REGION Network 7: Отключение
   RUNG wire#powerrail
      I_Contact( #Use.QF )
      wire#w1
      Coil( #xQF )
   END_RUNG
   RUNG wire#powerrail
      Contact( #CMD.Sim )
   END_RUNG wire#w1
   RUNG wire#powerrail
      Contact( #Use.QF )
      Contact( #FB.QF )
      I_Contact( #CMD.Sim )
   END_RUNG wire#w1
   RUNG wire#powerrail
      I_Contact( #Use.KM )
      Contact( #CMD.Start_M )
      I_Contact( #CMD.Sim )
      wire#w2
      Coil( #xKM )
   END_RUNG
   RUNG wire#powerrail
      Contact( #Use.KM )
      wire#w3
      Contact( #FB.KM )
   END_RUNG wire#w2
   RUNG wire#powerrail
      Contact( #CMD.Sim )
   END_RUNG wire#w3
   // the same network as SCL:
   #xQF := NOT #Use.QF OR #CMD.Sim OR (#Use.QF AND #FB.QF AND NOT #CMD.Sim);
   #xKM := (NOT #Use.KM AND #CMD.Start_M AND NOT #CMD.Sim) OR ((#Use.KM OR #CMD.Sim) AND #FB.KM);
END_REGION

REGION Network 8: Режим работы устройства / определение режима работы
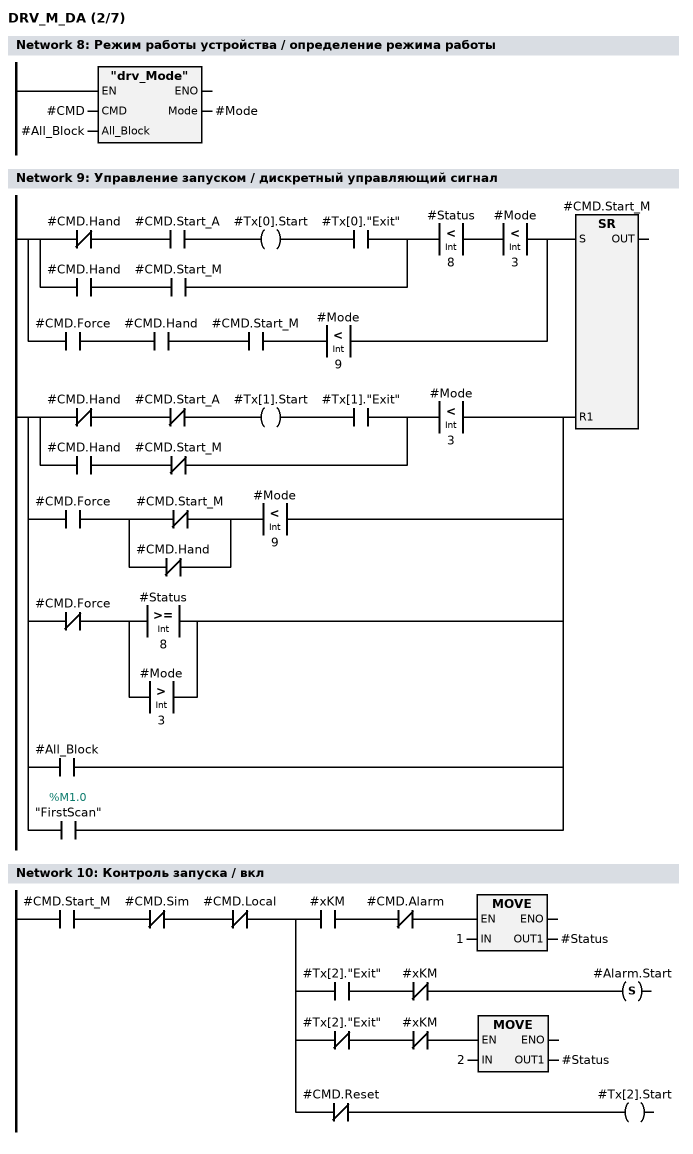
   RUNG wire#powerrail
      "drv_Mode"(CMD := #CMD, All_Block := #All_Block, Mode => #Mode)
   END_RUNG
   // the same network as SCL:
   "drv_Mode"(CMD := #CMD, All_Block := #All_Block, Mode => #Mode);
END_REGION

REGION Network 9: Управление запуском / дискретный управляющий сигнал
   RUNG wire#powerrail
      I_Contact( #CMD.Hand )
      Contact( #CMD.Start_A )
      Coil( #Tx[0].Start )
      Contact( #Tx[0]."Exit" )
      wire#w1
      { S7_Templates := "SrcType := Int" } LT_Contact(in1 := #Status, in2 := 8)
      { S7_Templates := "SrcType := Int" } LT_Contact(in1 := #Mode, in2 := 3)
      wire#w2
      S_SR(operand := #CMD.Start_M, r1 := wire#w7)
   END_RUNG
   RUNG wire#powerrail
      Contact( #CMD.Hand )
      Contact( #CMD.Start_M )
   END_RUNG wire#w1
   RUNG wire#powerrail
      Contact( #CMD.Force )
      Contact( #CMD.Hand )
      Contact( #CMD.Start_M )
      { S7_Templates := "SrcType := Int" } LT_Contact(in1 := #Mode, in2 := 9)
   END_RUNG wire#w2
   RUNG wire#powerrail
      I_Contact( #CMD.Hand )
      I_Contact( #CMD.Start_A )
      Coil( #Tx[1].Start )
      Contact( #Tx[1]."Exit" )
      wire#w3
      { S7_Templates := "SrcType := Int" } LT_Contact(in1 := #Mode, in2 := 3)
   END_RUNG wire#w7
   RUNG wire#powerrail
      Contact( #CMD.Hand )
      I_Contact( #CMD.Start_M )
   END_RUNG wire#w3
   RUNG wire#powerrail
      Contact( #CMD.Force )
      wire#w4
      I_Contact( #CMD.Start_M )
      wire#w5
      { S7_Templates := "SrcType := Int" } LT_Contact(in1 := #Mode, in2 := 9)
   END_RUNG wire#w7
   RUNG wire#w4
      I_Contact( #CMD.Hand )
   END_RUNG wire#w5
   RUNG wire#powerrail
      I_Contact( #CMD.Force )
      wire#w6
      { S7_Templates := "SrcType := Int" } GE_Contact(in1 := #Status, in2 := 8)
   END_RUNG wire#w7
   RUNG wire#w6
      { S7_Templates := "SrcType := Int" } GT_Contact(in1 := #Mode, in2 := 3)
   END_RUNG wire#w7
   RUNG wire#powerrail
      Contact( #All_Block )
   END_RUNG wire#w7
   RUNG wire#powerrail
      Contact( "FirstScan" )
   END_RUNG wire#w7
   // the same network as SCL:
   #Tx[0].Start := NOT #CMD.Hand AND #CMD.Start_A;
   #_w1 := (((NOT #CMD.Hand AND #CMD.Start_A AND #Tx[0]."Exit") OR (#CMD.Hand AND #CMD.Start_M)) AND (#Status < 8) AND (#Mode < 3)) OR (#CMD.Force AND #CMD.Hand AND #CMD.Start_M AND (#Mode < 9));
   #Tx[1].Start := NOT #CMD.Hand AND NOT #CMD.Start_A;
   #_w2 := (((NOT #CMD.Hand AND NOT #CMD.Start_A AND #Tx[1]."Exit") OR (#CMD.Hand AND NOT #CMD.Start_M)) AND (#Mode < 3)) OR (#CMD.Force AND (NOT #CMD.Start_M OR NOT #CMD.Hand) AND (#Mode < 9)) OR (NOT #CMD.Force AND ((#Status >= 8) OR (#Mode > 3))) OR #All_Block OR "FirstScan";
   IF #_w1 THEN
       #CMD.Start_M := TRUE;   // SR flip-flop
   END_IF;
   IF #_w2 THEN #CMD.Start_M := FALSE; END_IF;
END_REGION

REGION Network 10: Контроль запуска / вкл
   RUNG wire#powerrail
      Contact( #CMD.Start_M )
      I_Contact( #CMD.Sim )
      I_Contact( #CMD.Local )
      wire#w1
      Contact( #xKM )
      I_Contact( #CMD.Alarm )
      { S7_GenerateENO := "TRUE" } Move(in := 1, out1 => #Status)
   END_RUNG
   RUNG wire#w1
      Contact( #Tx[2]."Exit" )
      I_Contact( #xKM )
      S_Coil( #Alarm.Start )
   END_RUNG
   RUNG wire#w1
      I_Contact( #Tx[2]."Exit" )
      I_Contact( #xKM )
      { S7_GenerateENO := "TRUE" } Move(in := 2, out1 => #Status)
   END_RUNG
   RUNG wire#w1
      I_Contact( #CMD.Reset )
      Coil( #Tx[2].Start )
   END_RUNG
   // the same network as SCL:
   #_w1 := #CMD.Start_M AND NOT #CMD.Sim AND NOT #CMD.Local;
   IF #_w1 AND #xKM AND NOT #CMD.Alarm THEN #Status := 1; END_IF;
   IF #_w1 AND #Tx[2]."Exit" AND NOT #xKM THEN #Alarm.Start := TRUE; END_IF;
   IF #_w1 AND NOT #Tx[2]."Exit" AND NOT #xKM THEN #Status := 2; END_IF;
   #Tx[2].Start := #_w1 AND NOT #CMD.Reset;
END_REGION

REGION Network 11: Контроль останова / выкл
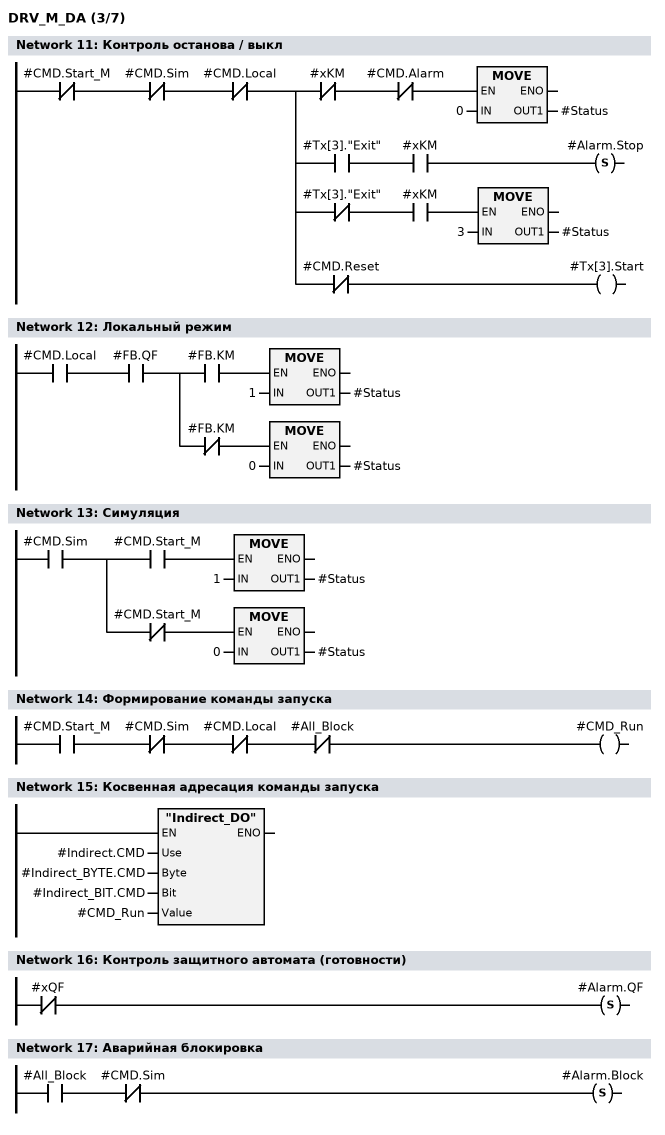
   RUNG wire#powerrail
      I_Contact( #CMD.Start_M )
      I_Contact( #CMD.Sim )
      I_Contact( #CMD.Local )
      wire#w1
      I_Contact( #xKM )
      I_Contact( #CMD.Alarm )
      { S7_GenerateENO := "TRUE" } Move(in := 0, out1 => #Status)
   END_RUNG
   RUNG wire#w1
      Contact( #Tx[3]."Exit" )
      Contact( #xKM )
      S_Coil( #Alarm.Stop )
   END_RUNG
   RUNG wire#w1
      I_Contact( #Tx[3]."Exit" )
      Contact( #xKM )
      { S7_GenerateENO := "TRUE" } Move(in := 3, out1 => #Status)
   END_RUNG
   RUNG wire#w1
      I_Contact( #CMD.Reset )
      Coil( #Tx[3].Start )
   END_RUNG
   // the same network as SCL:
   #_w1 := NOT #CMD.Start_M AND NOT #CMD.Sim AND NOT #CMD.Local;
   IF #_w1 AND NOT #xKM AND NOT #CMD.Alarm THEN #Status := 0; END_IF;
   IF #_w1 AND #Tx[3]."Exit" AND #xKM THEN #Alarm.Stop := TRUE; END_IF;
   IF #_w1 AND NOT #Tx[3]."Exit" AND #xKM THEN #Status := 3; END_IF;
   #Tx[3].Start := #_w1 AND NOT #CMD.Reset;
END_REGION

REGION Network 12: Локальный режим
   RUNG wire#powerrail
      Contact( #CMD.Local )
      Contact( #FB.QF )
      wire#w1
      Contact( #FB.KM )
      { S7_GenerateENO := "TRUE" } Move(in := 1, out1 => #Status)
   END_RUNG
   RUNG wire#w1
      I_Contact( #FB.KM )
      { S7_GenerateENO := "TRUE" } Move(in := 0, out1 => #Status)
   END_RUNG
   // the same network as SCL:
   #_w1 := #CMD.Local AND #FB.QF;
   IF #_w1 AND #FB.KM THEN #Status := 1; END_IF;
   IF #_w1 AND NOT #FB.KM THEN #Status := 0; END_IF;
END_REGION

REGION Network 13: Симуляция
   RUNG wire#powerrail
      Contact( #CMD.Sim )
      wire#w1
      Contact( #CMD.Start_M )
      { S7_GenerateENO := "TRUE" } Move(in := 1, out1 => #Status)
   END_RUNG
   RUNG wire#w1
      I_Contact( #CMD.Start_M )
      { S7_GenerateENO := "TRUE" } Move(in := 0, out1 => #Status)
   END_RUNG
   // the same network as SCL:
   IF #CMD.Sim AND #CMD.Start_M THEN #Status := 1; END_IF;
   IF #CMD.Sim AND NOT #CMD.Start_M THEN #Status := 0; END_IF;
END_REGION

REGION Network 14: Формирование команды запуска
   RUNG wire#powerrail
      Contact( #CMD.Start_M )
      I_Contact( #CMD.Sim )
      I_Contact( #CMD.Local )
      I_Contact( #All_Block )
      Coil( #CMD_Run )
   END_RUNG
   // the same network as SCL:
   #CMD_Run := #CMD.Start_M AND NOT #CMD.Sim AND NOT #CMD.Local AND NOT #All_Block;
END_REGION

REGION Network 15: Косвенная адресация команды запуска
   RUNG wire#powerrail
      "Indirect_DO"(Use := #Indirect.CMD, "Byte" := #Indirect_BYTE.CMD, Bit := #Indirect_BIT.CMD, Value := #CMD_Run)
   END_RUNG
   // the same network as SCL:
   "Indirect_DO"(Use := #Indirect.CMD,
                 "Byte" := #Indirect_BYTE.CMD,
                 Bit := #Indirect_BIT.CMD,
                 Value := #CMD_Run);
END_REGION

REGION Network 16: Контроль защитного автомата (готовности)
   RUNG wire#powerrail
      I_Contact( #xQF )
      S_Coil( #Alarm.QF )
   END_RUNG
   // the same network as SCL:
   IF NOT #xQF THEN #Alarm.QF := TRUE; END_IF;
END_REGION

REGION Network 17: Аварийная блокировка
   RUNG wire#powerrail
      Contact( #All_Block )
      I_Contact( #CMD.Sim )
      S_Coil( #Alarm.Block )
   END_RUNG
   // the same network as SCL:
   IF #All_Block AND NOT #CMD.Sim THEN #Alarm.Block := TRUE; END_IF;
END_REGION

REGION Network 18: Сигнал аварии
   // Safety - сработал датчик безопасности, подключается через отдельный дискретный вход
   // Termo - сработала термозащита, подключается через отдельный дискретный вход
   // Alarm - сработала внешняя авария, подключается через отдельный дискретный вход
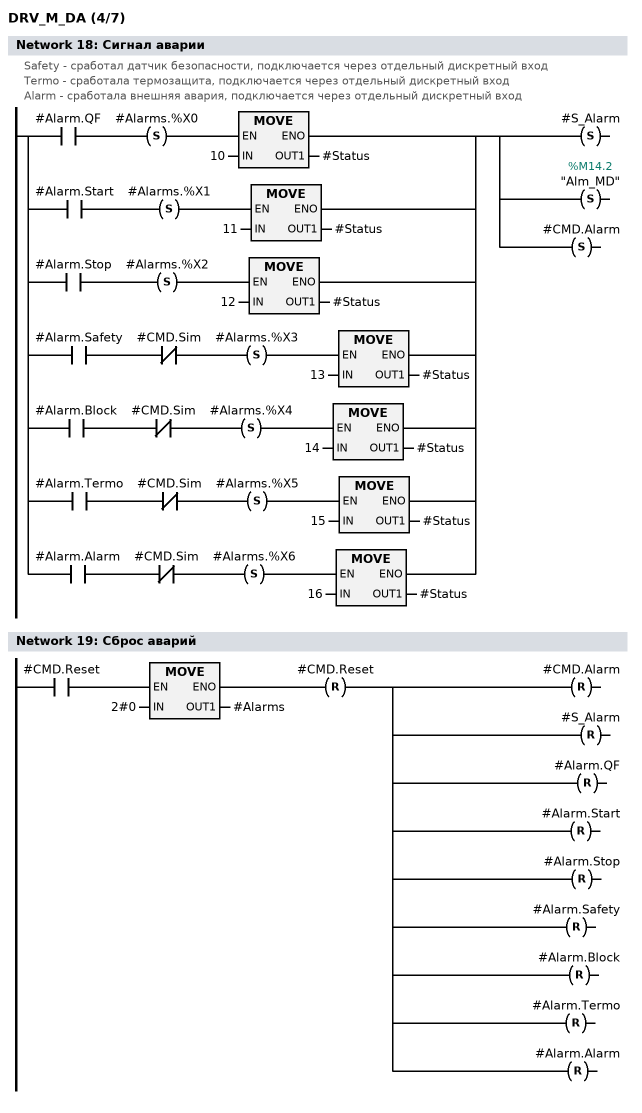
   RUNG wire#powerrail
      Contact( #Alarm.QF )
      S_Coil( #Alarms.%X0 )
      { S7_GenerateENO := "TRUE" } Move(in := 10, out1 => #Status)
      wire#w1
      S_Coil( #S_Alarm )
   END_RUNG
   RUNG wire#powerrail
      Contact( #Alarm.Start )
      S_Coil( #Alarms.%X1 )
      { S7_GenerateENO := "TRUE" } Move(in := 11, out1 => #Status)
   END_RUNG wire#w1
   RUNG wire#powerrail
      Contact( #Alarm.Stop )
      S_Coil( #Alarms.%X2 )
      { S7_GenerateENO := "TRUE" } Move(in := 12, out1 => #Status)
   END_RUNG wire#w1
   RUNG wire#powerrail
      Contact( #Alarm.Safety )
      I_Contact( #CMD.Sim )
      S_Coil( #Alarms.%X3 )
      { S7_GenerateENO := "TRUE" } Move(in := 13, out1 => #Status)
   END_RUNG wire#w1
   RUNG wire#powerrail
      Contact( #Alarm.Block )
      I_Contact( #CMD.Sim )
      S_Coil( #Alarms.%X4 )
      { S7_GenerateENO := "TRUE" } Move(in := 14, out1 => #Status)
   END_RUNG wire#w1
   RUNG wire#powerrail
      Contact( #Alarm.Termo )
      I_Contact( #CMD.Sim )
      S_Coil( #Alarms.%X5 )
      { S7_GenerateENO := "TRUE" } Move(in := 15, out1 => #Status)
   END_RUNG wire#w1
   RUNG wire#powerrail
      Contact( #Alarm.Alarm )
      I_Contact( #CMD.Sim )
      S_Coil( #Alarms.%X6 )
      { S7_GenerateENO := "TRUE" } Move(in := 16, out1 => #Status)
   END_RUNG wire#w1
   RUNG wire#w1
      S_Coil( "Alm_MD" )
   END_RUNG
   RUNG wire#w1
      S_Coil( #CMD.Alarm )
   END_RUNG
   // the same network as SCL:
   // ENO of a box is taken as its EN; it also drops when the box reports an error
   IF #Alarm.QF THEN
       #Alarms.%X0 := TRUE;
       #Status := 10;
   END_IF;
   IF #Alarm.Start THEN
       #Alarms.%X1 := TRUE;
       #Status := 11;
   END_IF;
   IF #Alarm.Stop THEN
       #Alarms.%X2 := TRUE;
       #Status := 12;
   END_IF;
   #_w1 := #Alarm.Safety AND NOT #CMD.Sim;
   IF #_w1 THEN
       #Alarms.%X3 := TRUE;
       #Status := 13;
   END_IF;
   #_w2 := #Alarm.Block AND NOT #CMD.Sim;
   IF #_w2 THEN
       #Alarms.%X4 := TRUE;
       #Status := 14;
   END_IF;
   #_w3 := #Alarm.Termo AND NOT #CMD.Sim;
   IF #_w3 THEN
       #Alarms.%X5 := TRUE;
       #Status := 15;
   END_IF;
   #_w4 := #Alarm.Alarm AND NOT #CMD.Sim;
   IF #_w4 THEN
       #Alarms.%X6 := TRUE;
       #Status := 16;
   END_IF;
   IF #Alarm.QF OR #Alarm.Start OR #Alarm.Stop OR #_w1 OR #_w2 OR #_w3 OR #_w4 THEN
       #S_Alarm := TRUE;
       "Alm_MD" := TRUE;
       #CMD.Alarm := TRUE;
   END_IF;
END_REGION

REGION Network 19: Сброс аварий
   RUNG wire#powerrail
      Contact( #CMD.Reset )
      Move(in := 2#0, out1 => #Alarms)
      R_Coil( #CMD.Reset )
      wire#w1
      R_Coil( #CMD.Alarm )
   END_RUNG
   RUNG wire#w1
      R_Coil( #S_Alarm )
   END_RUNG
   RUNG wire#w1
      R_Coil( #Alarm.QF )
   END_RUNG
   RUNG wire#w1
      R_Coil( #Alarm.Start )
   END_RUNG
   RUNG wire#w1
      R_Coil( #Alarm.Stop )
   END_RUNG
   RUNG wire#w1
      R_Coil( #Alarm.Safety )
   END_RUNG
   RUNG wire#w1
      R_Coil( #Alarm.Block )
   END_RUNG
   RUNG wire#w1
      R_Coil( #Alarm.Termo )
   END_RUNG
   RUNG wire#w1
      R_Coil( #Alarm.Alarm )
   END_RUNG
   // the same network as SCL:
   IF #CMD.Reset THEN #Alarms := 2#0; END_IF;
   #_w1 := #CMD.Reset;
   IF #_w1 THEN
       #CMD.Reset := FALSE;
       #CMD.Alarm := FALSE;
       #S_Alarm := FALSE;
       #Alarm.QF := FALSE;
       #Alarm.Start := FALSE;
       #Alarm.Stop := FALSE;
       #Alarm.Safety := FALSE;
       #Alarm.Block := FALSE;
       #Alarm.Termo := FALSE;
       #Alarm.Alarm := FALSE;
   END_IF;
END_REGION

REGION Network 20: События привода
   // 0 - ручной режим активирован
   // 1 - ручной режим деактивирован
   // 2 - принудительный режим активирован
   // 3 - принудительный режим деактивирован
   // 4 - запуск в ручном режиме
   // 5 - останов в ручном режиме
   // 6 - местный режим управления активирован
   // 7 - местный режим управления деактивирован
   // 8 - запущено в местном режиме
   // 9 - остановлено в местном режиме
   // 10 - сервисный режим активирован
   // 11 - сервисный режим деактивирован
   // 12 - проведено сервисное обслуживание
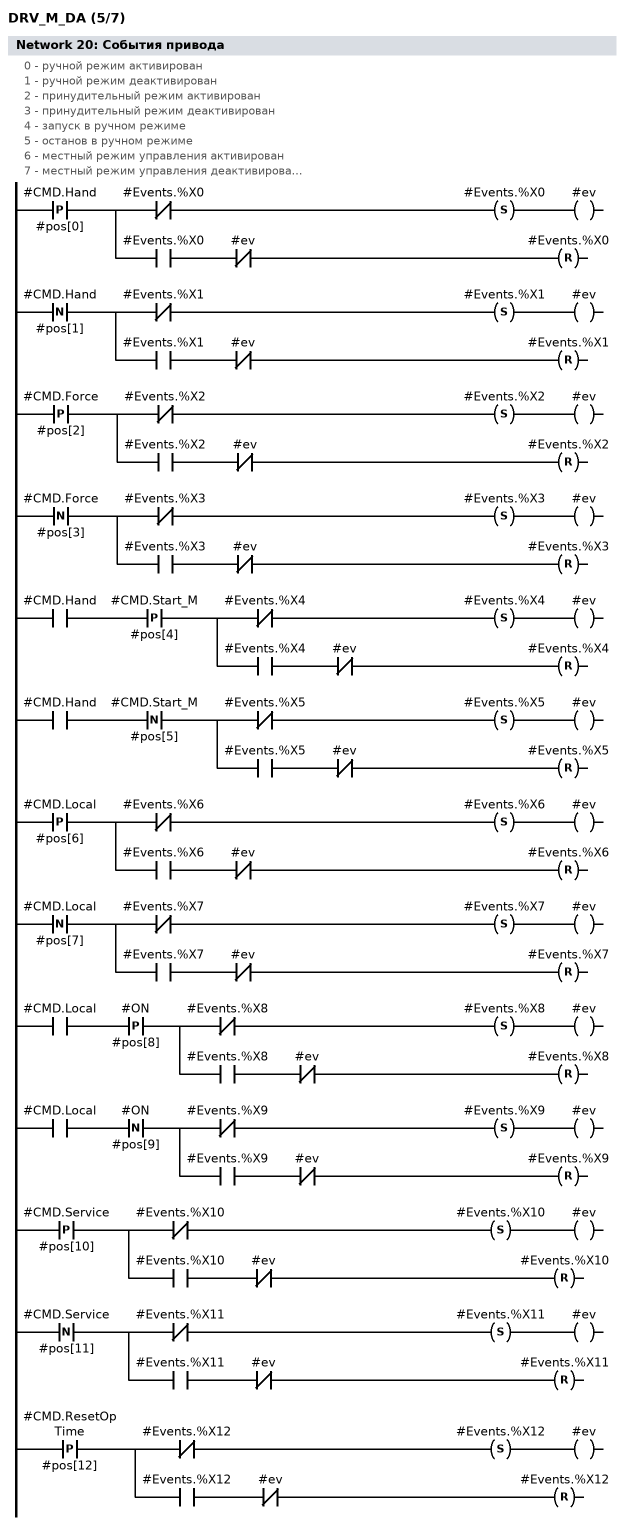
   RUNG wire#powerrail
      P_Contact(operand := #CMD.Hand, bit := #pos[0])
      wire#w1
      I_Contact( #Events.%X0 )
      S_Coil( #Events.%X0 )
      Coil( #ev )
   END_RUNG
   RUNG wire#w1
      Contact( #Events.%X0 )
      I_Contact( #ev )
      R_Coil( #Events.%X0 )
   END_RUNG
   RUNG wire#powerrail
      N_Contact(operand := #CMD.Hand, bit := #pos[1])
      wire#w2
      I_Contact( #Events.%X1 )
      S_Coil( #Events.%X1 )
      Coil( #ev )
   END_RUNG
   RUNG wire#w2
      Contact( #Events.%X1 )
      I_Contact( #ev )
      R_Coil( #Events.%X1 )
   END_RUNG
   RUNG wire#powerrail
      P_Contact(operand := #CMD.Force, bit := #pos[2])
      wire#w3
      I_Contact( #Events.%X2 )
      S_Coil( #Events.%X2 )
      Coil( #ev )
   END_RUNG
   RUNG wire#w3
      Contact( #Events.%X2 )
      I_Contact( #ev )
      R_Coil( #Events.%X2 )
   END_RUNG
   RUNG wire#powerrail
      N_Contact(operand := #CMD.Force, bit := #pos[3])
      wire#w4
      I_Contact( #Events.%X3 )
      S_Coil( #Events.%X3 )
      Coil( #ev )
   END_RUNG
   RUNG wire#w4
      Contact( #Events.%X3 )
      I_Contact( #ev )
      R_Coil( #Events.%X3 )
   END_RUNG
   RUNG wire#powerrail
      Contact( #CMD.Hand )
      P_Contact(operand := #CMD.Start_M, bit := #pos[4])
      wire#w5
      I_Contact( #Events.%X4 )
      S_Coil( #Events.%X4 )
      Coil( #ev )
   END_RUNG
   RUNG wire#w5
      Contact( #Events.%X4 )
      I_Contact( #ev )
      R_Coil( #Events.%X4 )
   END_RUNG
   RUNG wire#powerrail
      Contact( #CMD.Hand )
      N_Contact(operand := #CMD.Start_M, bit := #pos[5])
      wire#w6
      I_Contact( #Events.%X5 )
      S_Coil( #Events.%X5 )
      Coil( #ev )
   END_RUNG
   RUNG wire#w6
      Contact( #Events.%X5 )
      I_Contact( #ev )
      R_Coil( #Events.%X5 )
   END_RUNG
   RUNG wire#powerrail
      P_Contact(operand := #CMD.Local, bit := #pos[6])
      wire#w7
      I_Contact( #Events.%X6 )
      S_Coil( #Events.%X6 )
      Coil( #ev )
   END_RUNG
   RUNG wire#w7
      Contact( #Events.%X6 )
      I_Contact( #ev )
      R_Coil( #Events.%X6 )
   END_RUNG
   RUNG wire#powerrail
      N_Contact(operand := #CMD.Local, bit := #pos[7])
      wire#w8
      I_Contact( #Events.%X7 )
      S_Coil( #Events.%X7 )
      Coil( #ev )
   END_RUNG
   RUNG wire#w8
      Contact( #Events.%X7 )
      I_Contact( #ev )
      R_Coil( #Events.%X7 )
   END_RUNG
   RUNG wire#powerrail
      Contact( #CMD.Local )
      P_Contact(operand := #ON, bit := #pos[8])
      wire#w9
      I_Contact( #Events.%X8 )
      S_Coil( #Events.%X8 )
      Coil( #ev )
   END_RUNG
   RUNG wire#w9
      Contact( #Events.%X8 )
      I_Contact( #ev )
      R_Coil( #Events.%X8 )
   END_RUNG
   RUNG wire#powerrail
      Contact( #CMD.Local )
      N_Contact(operand := #ON, bit := #pos[9])
      wire#w10
      I_Contact( #Events.%X9 )
      S_Coil( #Events.%X9 )
      Coil( #ev )
   END_RUNG
   RUNG wire#w10
      Contact( #Events.%X9 )
      I_Contact( #ev )
      R_Coil( #Events.%X9 )
   END_RUNG
   RUNG wire#powerrail
      P_Contact(operand := #CMD.Service, bit := #pos[10])
      wire#w11
      I_Contact( #Events.%X10 )
      S_Coil( #Events.%X10 )
      Coil( #ev )
   END_RUNG
   RUNG wire#w11
      Contact( #Events.%X10 )
      I_Contact( #ev )
      R_Coil( #Events.%X10 )
   END_RUNG
   RUNG wire#powerrail
      N_Contact(operand := #CMD.Service, bit := #pos[11])
      wire#w12
      I_Contact( #Events.%X11 )
      S_Coil( #Events.%X11 )
      Coil( #ev )
   END_RUNG
   RUNG wire#w12
      Contact( #Events.%X11 )
      I_Contact( #ev )
      R_Coil( #Events.%X11 )
   END_RUNG
   RUNG wire#powerrail
      P_Contact(operand := #CMD.ResetOpTime, bit := #pos[12])
      wire#w13
      I_Contact( #Events.%X12 )
      S_Coil( #Events.%X12 )
      Coil( #ev )
   END_RUNG
   RUNG wire#w13
      Contact( #Events.%X12 )
      I_Contact( #ev )
      R_Coil( #Events.%X12 )
   END_RUNG
   // the same network as SCL:
   #_w1 := #CMD.Hand AND NOT #pos[0];   // rising edge of #CMD.Hand
   #pos[0] := #CMD.Hand;
   #_w2 := #_w1 AND NOT #Events.%X0;
   IF #_w2 THEN #Events.%X0 := TRUE; END_IF;
   #ev := #_w2;
   IF #_w1 AND #Events.%X0 AND NOT #ev THEN #Events.%X0 := FALSE; END_IF;
   #_w3 := NOT #CMD.Hand AND #pos[1];   // falling edge of #CMD.Hand
   #pos[1] := #CMD.Hand;
   #_w4 := #_w3 AND NOT #Events.%X1;
   IF #_w4 THEN #Events.%X1 := TRUE; END_IF;
   #ev := #_w4;
   IF #_w3 AND #Events.%X1 AND NOT #ev THEN #Events.%X1 := FALSE; END_IF;
   #_w5 := #CMD.Force AND NOT #pos[2];   // rising edge of #CMD.Force
   #pos[2] := #CMD.Force;
   #_w6 := #_w5 AND NOT #Events.%X2;
   IF #_w6 THEN #Events.%X2 := TRUE; END_IF;
   #ev := #_w6;
   IF #_w5 AND #Events.%X2 AND NOT #ev THEN #Events.%X2 := FALSE; END_IF;
   #_w7 := NOT #CMD.Force AND #pos[3];   // falling edge of #CMD.Force
   #pos[3] := #CMD.Force;
   #_w8 := #_w7 AND NOT #Events.%X3;
   IF #_w8 THEN #Events.%X3 := TRUE; END_IF;
   #ev := #_w8;
   IF #_w7 AND #Events.%X3 AND NOT #ev THEN #Events.%X3 := FALSE; END_IF;
   #_w9 := #CMD.Hand AND #CMD.Start_M AND NOT #pos[4];   // rising edge of #CMD.Start_M
   #pos[4] := #CMD.Start_M;
   #_w10 := #_w9 AND NOT #Events.%X4;
   IF #_w10 THEN #Events.%X4 := TRUE; END_IF;
   #ev := #_w10;
   IF #_w9 AND #Events.%X4 AND NOT #ev THEN #Events.%X4 := FALSE; END_IF;
   #_w11 := #CMD.Hand AND NOT #CMD.Start_M AND #pos[5];   // falling edge of #CMD.Start_M
   #pos[5] := #CMD.Start_M;
   #_w12 := #_w11 AND NOT #Events.%X5;
   IF #_w12 THEN #Events.%X5 := TRUE; END_IF;
   #ev := #_w12;
   IF #_w11 AND #Events.%X5 AND NOT #ev THEN #Events.%X5 := FALSE; END_IF;
   #_w13 := #CMD.Local AND NOT #pos[6];   // rising edge of #CMD.Local
   #pos[6] := #CMD.Local;
   #_w14 := #_w13 AND NOT #Events.%X6;
   IF #_w14 THEN #Events.%X6 := TRUE; END_IF;
   #ev := #_w14;
   IF #_w13 AND #Events.%X6 AND NOT #ev THEN #Events.%X6 := FALSE; END_IF;
   #_w15 := NOT #CMD.Local AND #pos[7];   // falling edge of #CMD.Local
   #pos[7] := #CMD.Local;
   #_w16 := #_w15 AND NOT #Events.%X7;
   IF #_w16 THEN #Events.%X7 := TRUE; END_IF;
   #ev := #_w16;
   IF #_w15 AND #Events.%X7 AND NOT #ev THEN #Events.%X7 := FALSE; END_IF;
   #_w17 := #CMD.Local AND #ON AND NOT #pos[8];   // rising edge of #ON
   #pos[8] := #ON;
   #_w18 := #_w17 AND NOT #Events.%X8;
   IF #_w18 THEN #Events.%X8 := TRUE; END_IF;
   #ev := #_w18;
   IF #_w17 AND #Events.%X8 AND NOT #ev THEN #Events.%X8 := FALSE; END_IF;
   #_w19 := #CMD.Local AND NOT #ON AND #pos[9];   // falling edge of #ON
   #pos[9] := #ON;
   #_w20 := #_w19 AND NOT #Events.%X9;
   IF #_w20 THEN #Events.%X9 := TRUE; END_IF;
   #ev := #_w20;
   IF #_w19 AND #Events.%X9 AND NOT #ev THEN #Events.%X9 := FALSE; END_IF;
   #_w21 := #CMD.Service AND NOT #pos[10];   // rising edge of #CMD.Service
   #pos[10] := #CMD.Service;
   #_w22 := #_w21 AND NOT #Events.%X10;
   IF #_w22 THEN #Events.%X10 := TRUE; END_IF;
   #ev := #_w22;
   IF #_w21 AND #Events.%X10 AND NOT #ev THEN #Events.%X10 := FALSE; END_IF;
   #_w23 := NOT #CMD.Service AND #pos[11];   // falling edge of #CMD.Service
   #pos[11] := #CMD.Service;
   #_w24 := #_w23 AND NOT #Events.%X11;
   IF #_w24 THEN #Events.%X11 := TRUE; END_IF;
   #ev := #_w24;
   IF #_w23 AND #Events.%X11 AND NOT #ev THEN #Events.%X11 := FALSE; END_IF;
   #_w25 := #CMD.ResetOpTime AND NOT #pos[12];   // rising edge of #CMD.ResetOpTime
   #pos[12] := #CMD.ResetOpTime;
   #_w26 := #_w25 AND NOT #Events.%X12;
   IF #_w26 THEN #Events.%X12 := TRUE; END_IF;
   #ev := #_w26;
   IF #_w25 AND #Events.%X12 AND NOT #ev THEN #Events.%X12 := FALSE; END_IF;
END_REGION

REGION Network 21: Сервисный режим
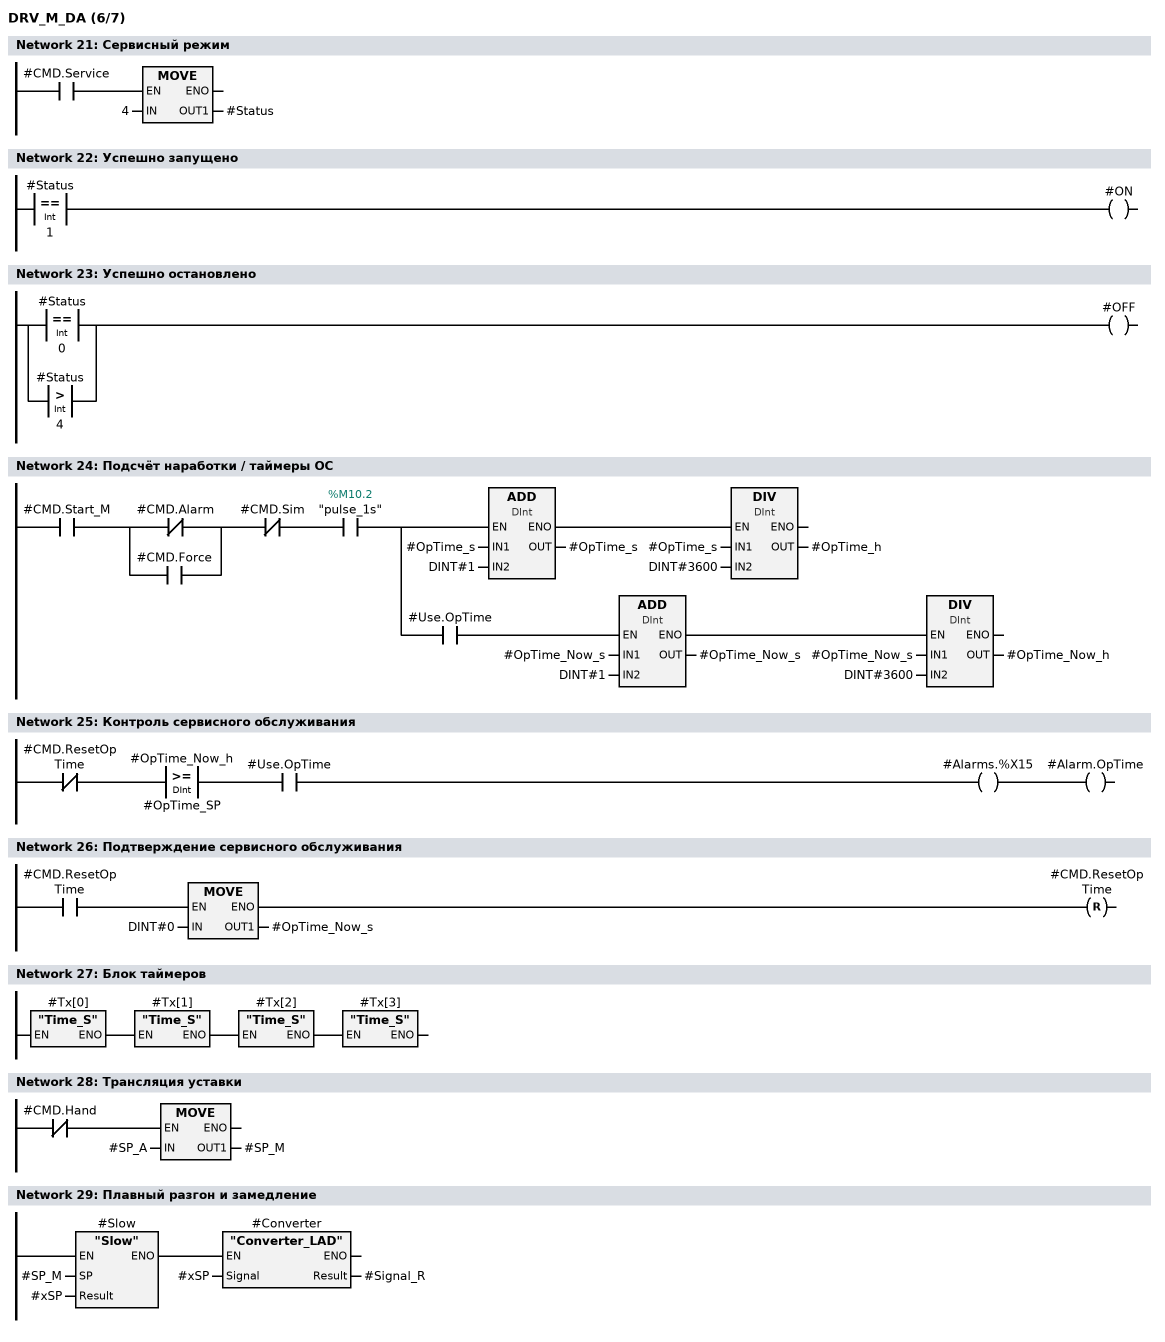
   RUNG wire#powerrail
      Contact( #CMD.Service )
      { S7_GenerateENO := "TRUE" } Move(in := 4, out1 => #Status)
   END_RUNG
   // the same network as SCL:
   IF #CMD.Service THEN #Status := 4; END_IF;
END_REGION

REGION Network 22: Успешно запущено
   RUNG wire#powerrail
      { S7_Templates := "SrcType := Int" } EQ_Contact(in1 := #Status, in2 := 1)
      Coil( #ON )
   END_RUNG
   // the same network as SCL:
   #ON := #Status = 1;
END_REGION

REGION Network 23: Успешно остановлено
   RUNG wire#powerrail
      { S7_Templates := "SrcType := Int" } EQ_Contact(in1 := #Status, in2 := 0)
      wire#w1
      Coil( #OFF )
   END_RUNG
   RUNG wire#powerrail
      { S7_Templates := "SrcType := Int" } GT_Contact(in1 := #Status, in2 := 4)
   END_RUNG wire#w1
   // the same network as SCL:
   #OFF := (#Status = 0) OR (#Status > 4);
END_REGION

REGION Network 24: Подсчёт наработки / таймеры ОС
   RUNG wire#powerrail
      Contact( #CMD.Start_M )
      wire#w1
      I_Contact( #CMD.Alarm )
      wire#w2
      I_Contact( #CMD.Sim )
      Contact( "pulse_1s" )
      wire#w3
      { S7_Templates := "SrcType := DInt"; S7_GenerateENO := "TRUE" } Add(in1 := #OpTime_s, in2 := DINT#1, out => #OpTime_s)
      { S7_Templates := "SrcType := DInt"; S7_GenerateENO := "TRUE" } Div(in1 := #OpTime_s, in2 := DINT#3600, out => #OpTime_h)
   END_RUNG
   RUNG wire#w1
      Contact( #CMD.Force )
   END_RUNG wire#w2
   RUNG wire#w3
      Contact( #Use.OpTime )
      { S7_Templates := "SrcType := DInt"; S7_GenerateENO := "TRUE" } Add(in1 := #OpTime_Now_s, in2 := DINT#1, out => #OpTime_Now_s)
      { S7_Templates := "SrcType := DInt"; S7_GenerateENO := "TRUE" } Div(in1 := #OpTime_Now_s, in2 := DINT#3600, out => #OpTime_Now_h)
   END_RUNG
   // the same network as SCL:
   // ENO of a box is taken as its EN; it also drops when the box reports an error
   #_w1 := #CMD.Start_M AND (NOT #CMD.Alarm OR #CMD.Force) AND NOT #CMD.Sim AND "pulse_1s";
   IF #_w1 THEN
       #OpTime_s := #OpTime_s + DINT#1;
       #OpTime_h := #OpTime_s / DINT#3600;
   END_IF;
   IF #_w1 AND #Use.OpTime THEN
       #OpTime_Now_s := #OpTime_Now_s + DINT#1;
       #OpTime_Now_h := #OpTime_Now_s / DINT#3600;
   END_IF;
END_REGION

REGION Network 25: Контроль сервисного обслуживания
   RUNG wire#powerrail
      I_Contact( #CMD.ResetOpTime )
      { S7_Templates := "SrcType := DInt" } GE_Contact(in1 := #OpTime_Now_h, in2 := #OpTime_SP)
      Contact( #Use.OpTime )
      Coil( #Alarms.%X15 )
      Coil( #Alarm.OpTime )
   END_RUNG
   // the same network as SCL:
   #Alarms.%X15 := NOT #CMD.ResetOpTime AND (#OpTime_Now_h >= #OpTime_SP) AND #Use.OpTime;
   #Alarm.OpTime := #Alarms.%X15;
END_REGION

REGION Network 26: Подтверждение сервисного обслуживания
   RUNG wire#powerrail
      Contact( #CMD.ResetOpTime )
      { S7_GenerateENO := "TRUE" } Move(in := DINT#0, out1 => #OpTime_Now_s)
      R_Coil( #CMD.ResetOpTime )
   END_RUNG
   // the same network as SCL:
   // ENO of a box is taken as its EN; it also drops when the box reports an error
   IF #CMD.ResetOpTime THEN
       #OpTime_Now_s := DINT#0;
       #CMD.ResetOpTime := FALSE;
   END_IF;
END_REGION

REGION Network 27: Блок таймеров
   RUNG wire#powerrail
      #Tx[0]()
      #Tx[1]()
      #Tx[2]()
      #Tx[3]()
   END_RUNG
   // the same network as SCL:
   #Tx[0](ENO => #_w1);   // "Time_S"
   #Tx[1](EN := #_w1, ENO => #_w2);   // "Time_S"
   #Tx[2](EN := #_w2, ENO => #_w3);   // "Time_S"
   IF #_w3 THEN
       #Tx[3]();   // "Time_S"
   END_IF;
END_REGION

REGION Network 28: Трансляция уставки
   RUNG wire#powerrail
      I_Contact( #CMD.Hand )
      Move(in := #SP_A, out1 => #SP_M)
   END_RUNG
   // the same network as SCL:
   IF NOT #CMD.Hand THEN #SP_M := #SP_A; END_IF;
END_REGION

REGION Network 29: Плавный разгон и замедление
   RUNG wire#powerrail
      #Slow(SP := #SP_M, Result := #xSP)
      #Converter(Signal := #xSP, Result => #Signal_R)
   END_RUNG
   // the same network as SCL:
   #Slow(SP := #SP_M, Result := #xSP, ENO => #_w1);   // "Slow"
   IF #_w1 THEN
       #Converter(Signal := #xSP, Result => #Signal_R);   // "Converter_LAD"
   END_IF;
END_REGION

REGION Network 30: Выходной аналоговый сигнал
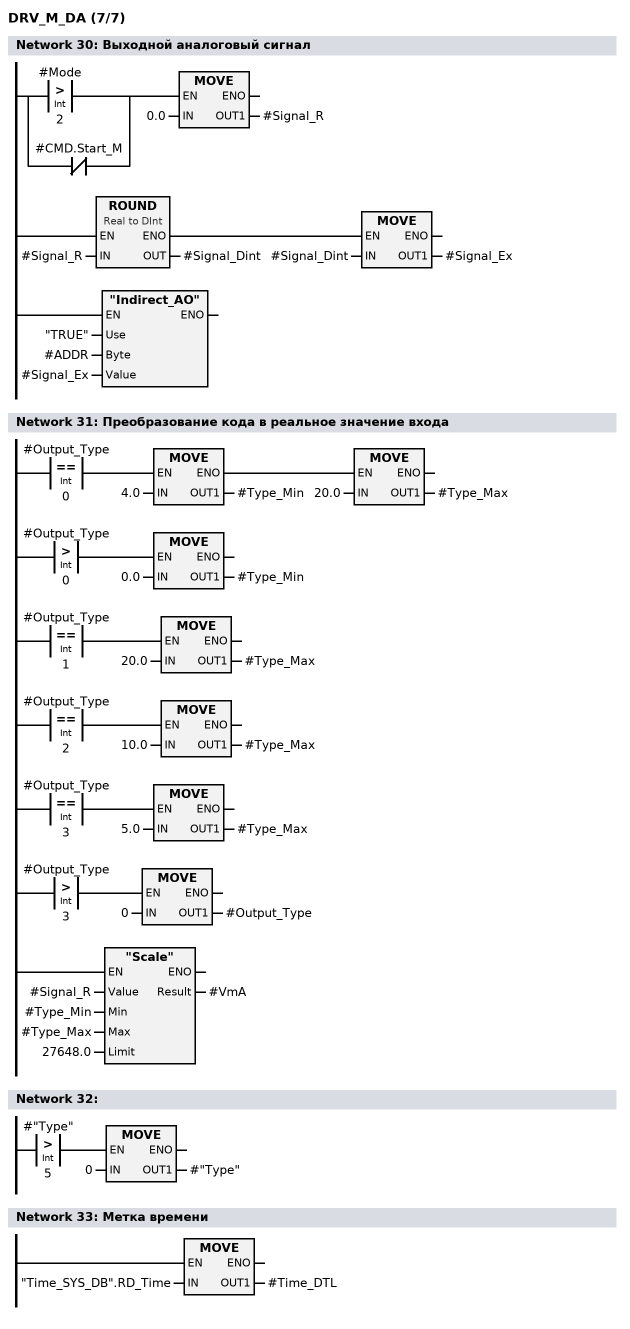
   RUNG wire#powerrail
      { S7_Templates := "SrcType := Int" } GT_Contact(in1 := #Mode, in2 := 2)
      wire#w1
      Move(in := 0.0, out1 => #Signal_R)
   END_RUNG
   RUNG wire#powerrail
      I_Contact( #CMD.Start_M )
   END_RUNG wire#w1
   RUNG wire#powerrail
      { S7_Templates := "[SrcType := Real, DestType := DInt]"; S7_GenerateENO := "TRUE" } Round(in := #Signal_R, out => #Signal_Dint)
      Move(in := #Signal_Dint, out1 => #Signal_Ex)
   END_RUNG
   RUNG wire#powerrail
      "Indirect_AO"(Use := "TRUE", "Byte" := #ADDR, Value := #Signal_Ex)
   END_RUNG
   // the same network as SCL:
   // ENO of a box is taken as its EN; it also drops when the box reports an error
   IF (#Mode > 2) OR NOT #CMD.Start_M THEN #Signal_R := 0.0; END_IF;
   #Signal_Dint := ROUND(#Signal_R);
   #Signal_Ex := #Signal_Dint;
   "Indirect_AO"(Use := "TRUE", "Byte" := #ADDR, Value := #Signal_Ex);
END_REGION

REGION Network 31: Преобразование кода в реальное значение входа
   RUNG wire#powerrail
      { S7_Templates := "SrcType := Int" } EQ_Contact(in1 := #Output_Type, in2 := 0)
      Move(in := 4.0, out1 => #Type_Min)
      Move(in := 20.0, out1 => #Type_Max)
   END_RUNG
   RUNG wire#powerrail
      { S7_Templates := "SrcType := Int" } GT_Contact(in1 := #Output_Type, in2 := 0)
      Move(in := 0.0, out1 => #Type_Min)
   END_RUNG
   RUNG wire#powerrail
      { S7_Templates := "SrcType := Int" } EQ_Contact(in1 := #Output_Type, in2 := 1)
      Move(in := 20.0, out1 => #Type_Max)
   END_RUNG
   RUNG wire#powerrail
      { S7_Templates := "SrcType := Int" } EQ_Contact(in1 := #Output_Type, in2 := 2)
      Move(in := 10.0, out1 => #Type_Max)
   END_RUNG
   RUNG wire#powerrail
      { S7_Templates := "SrcType := Int" } EQ_Contact(in1 := #Output_Type, in2 := 3)
      Move(in := 5.0, out1 => #Type_Max)
   END_RUNG
   RUNG wire#powerrail
      { S7_Templates := "SrcType := Int" } GT_Contact(in1 := #Output_Type, in2 := 3)
      Move(in := 0, out1 => #Output_Type)
   END_RUNG
   RUNG wire#powerrail
      "Scale"(Value := #Signal_R, Min := #Type_Min, Max := #Type_Max, Limit := 27648.0, Result => #VmA)
   END_RUNG
   // the same network as SCL:
   IF #Output_Type = 0 THEN
       #Type_Min := 4.0;
       #Type_Max := 20.0;
   END_IF;
   IF #Output_Type > 0 THEN #Type_Min := 0.0; END_IF;
   IF #Output_Type = 1 THEN #Type_Max := 20.0; END_IF;
   IF #Output_Type = 2 THEN #Type_Max := 10.0; END_IF;
   IF #Output_Type = 3 THEN #Type_Max := 5.0; END_IF;
   IF #Output_Type > 3 THEN #Output_Type := 0; END_IF;
   "Scale"(Value := #Signal_R, Min := #Type_Min, Max := #Type_Max, Limit := 27648.0, Result => #VmA);
END_REGION

REGION Network 32
   RUNG wire#powerrail
      { S7_Templates := "SrcType := Int" } GT_Contact(in1 := #"Type", in2 := 5)
      Move(in := 0, out1 => #"Type")
   END_RUNG
   // the same network as SCL:
   IF #"Type" > 5 THEN #"Type" := 0; END_IF;
END_REGION

REGION Network 33: Метка времени
   RUNG wire#powerrail
      Move(in := "Time_SYS_DB".RD_Time, out1 => #Time_DTL)
   END_RUNG
   // the same network as SCL:
   #Time_DTL := "Time_SYS_DB".RD_Time;
END_REGION
END_FUNCTION_BLOCK

FUNCTION_BLOCK "Valves"   // FB250, LAD
TITLE = Клапана
{ S7_Optimized_Access := 'FALSE' }
VERSION : 0.1
// FB_Alarm - аварийный сигнал для отключения клапана (например по давлению воздуха), 0 - авария, 1 - норма
// FB_QF - сигнал готовности к работе (например, по наличию 24в в линии управления пневмораспределителем), 0 - авария, 1 - норма
// FB_Open - обратная связь датчика открытия клапана, 0 - закрыт, 1 - открыт
// FB_Close - обратная связь датчика закрытия клапана, 1 - закрыт, 0 - открыт
// Value - управление аналоговым клапаном с позиционированием, формат Real, передаётся в блок AO_ex для конвертации в выходной сигнал контроллера (PQW), для использования установите #CMD.Analog в True
// 
// Q -  постоянный сигнал управления клапаном, 0 - закрыть, 1 - открыть
// stored: AutoNumber false, IsIECCheckEnabled false, SetENOAutomatically false, UDAEnableTagReadback false
   VAR DB_SPECIFIC
      Time_DTL { S7_SetPoint := 'True'} : DTL;
   END_VAR
BEGIN

REGION Network 1: Метка времени
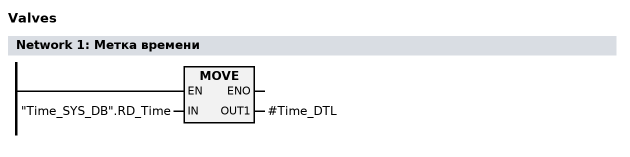
   RUNG wire#powerrail
      Move(in := "Time_SYS_DB".RD_Time, out1 => #Time_DTL)
   END_RUNG
   // the same network as SCL:
   #Time_DTL := "Time_SYS_DB".RD_Time;
END_REGION
END_FUNCTION_BLOCK

FUNCTION_BLOCK "Put_Get"   // FB2, LAD
TITLE = ADDR - удаленный PLC
{ S7_Optimized_Access := 'TRUE' }
VERSION : 0.1
// RD - блок в этом PLC
// stored: AutoNumber true, IsIECCheckEnabled false, IsRetainMemResEnabled false, MemoryReserve 100, SetENOAutomatically false, UDAEnableTagReadback false
   VAR
      GET_SKV_1 { S7_SetPoint := 'True'} : GET;
      GET_SKV_2 { S7_SetPoint := 'True'} : GET;
      GET_SKV_3 { S7_SetPoint := 'True'} : GET;
      GET_SKV_12 { S7_SetPoint := 'True'} : GET;
      GET_SKV_13 { S7_SetPoint := 'True'} : GET;
      GET_SKV_14 { S7_SetPoint := 'True'} : GET;
      GET_SKV_15 { S7_SetPoint := 'True'} : GET;
      GET_SKV_20 { S7_SetPoint := 'True'} : GET;
      GET_SKV_21 { S7_SetPoint := 'True'} : GET;
      GET_SKV_22 { S7_SetPoint := 'True'} : GET;
      GET_SKV_23 { S7_SetPoint := 'True'} : GET;
      PUT_SKV_1 { S7_SetPoint := 'True'} : PUT;
      PUT_SKV_2 { S7_SetPoint := 'True'} : PUT;
      PUT_SKV_3 { S7_SetPoint := 'True'} : PUT;
      PUT_SKV_12 { S7_SetPoint := 'True'} : PUT;
      PUT_SKV_13 { S7_SetPoint := 'True'} : PUT;
      PUT_SKV_14 { S7_SetPoint := 'True'} : PUT;
      PUT_SKV_15 { S7_SetPoint := 'True'} : PUT;
      PUT_SKV_20 { S7_SetPoint := 'True'} : PUT;
      PUT_SKV_21 { S7_SetPoint := 'True'} : PUT;
      PUT_SKV_22 { S7_SetPoint := 'True'} : PUT;
      PUT_SKV_23 { S7_SetPoint := 'True'} : PUT;
      GET_SKD2 { S7_SetPoint := 'True'} : GET;
      PUT_SKD2 { S7_SetPoint := 'True'} : PUT;
   END_VAR
   VAR_TEMP   // added for the SCL form of the ladder/FBD networks
      _w1 : Bool;
      _w2 : Bool;
   END_VAR
BEGIN

REGION Network 1: SKV 1
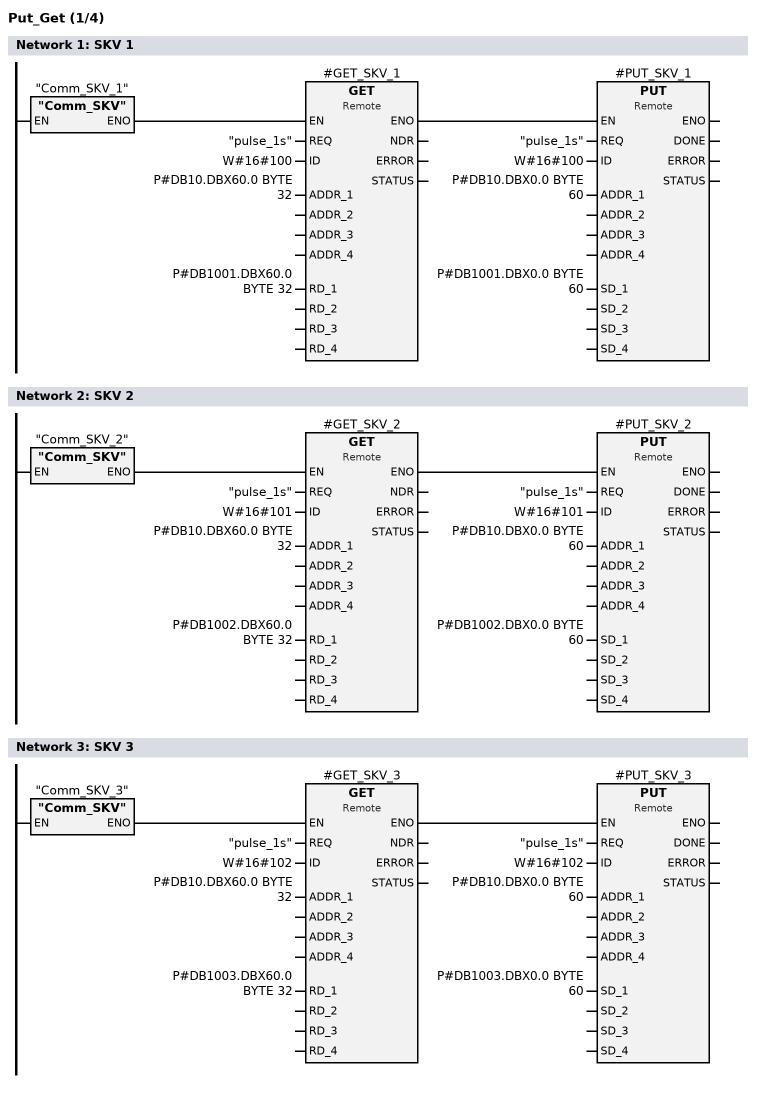
   RUNG wire#powerrail
      "Comm_SKV_1"()
      { S7_Templates := "[remote_type := Remote, local_type := Variant]" } #GET_SKV_1.GET(REQ := "pulse_1s", ID := W#16#100, ADDR_1 := P#DB10.DBX60.0 BYTE 32, ADDR_2 :=, ADDR_3 :=, ADDR_4 :=, RD_1 := P#DB1001.DBX60.0 BYTE 32, RD_2 :=, RD_3 :=, RD_4 :=, NDR =>, ERROR =>, STATUS =>)
      { S7_Templates := "[remote_type := Remote, local_type := Variant]" } #PUT_SKV_1.PUT(REQ := "pulse_1s", ID := W#16#100, ADDR_1 := P#DB10.DBX0.0 BYTE 60, ADDR_2 :=, ADDR_3 :=, ADDR_4 :=, SD_1 := P#DB1001.DBX0.0 BYTE 60, SD_2 :=, SD_3 :=, SD_4 :=, DONE =>, ERROR =>, STATUS =>)
   END_RUNG
   // the same network as SCL:
   "Comm_SKV_1"(ENO => #_w1);   // "Comm_SKV"
   #GET_SKV_1(EN := #_w1,   // GET
              REQ := "pulse_1s",
              ID := W#16#100,
              ADDR_1 := P#DB10.DBX60.0 BYTE 32,
              RD_1 := P#DB1001.DBX60.0 BYTE 32,
              ENO => #_w2);
   IF #_w2 THEN
       #PUT_SKV_1(REQ := "pulse_1s",   // PUT
                  ID := W#16#100,
                  ADDR_1 := P#DB10.DBX0.0 BYTE 60,
                  SD_1 := P#DB1001.DBX0.0 BYTE 60);
   END_IF;
END_REGION

REGION Network 2: SKV 2
   RUNG wire#powerrail
      "Comm_SKV_2"()
      { S7_Templates := "[remote_type := Remote, local_type := Variant]" } #GET_SKV_2.GET(REQ := "pulse_1s", ID := W#16#101, ADDR_1 := P#DB10.DBX60.0 BYTE 32, ADDR_2 :=, ADDR_3 :=, ADDR_4 :=, RD_1 := P#DB1002.DBX60.0 BYTE 32, RD_2 :=, RD_3 :=, RD_4 :=, NDR =>, ERROR =>, STATUS =>)
      { S7_Templates := "[remote_type := Remote, local_type := Variant]" } #PUT_SKV_2.PUT(REQ := "pulse_1s", ID := W#16#101, ADDR_1 := P#DB10.DBX0.0 BYTE 60, ADDR_2 :=, ADDR_3 :=, ADDR_4 :=, SD_1 := P#DB1002.DBX0.0 BYTE 60, SD_2 :=, SD_3 :=, SD_4 :=, DONE =>, ERROR =>, STATUS =>)
   END_RUNG
   // the same network as SCL:
   "Comm_SKV_2"(ENO => #_w1);   // "Comm_SKV"
   #GET_SKV_2(EN := #_w1,   // GET
              REQ := "pulse_1s",
              ID := W#16#101,
              ADDR_1 := P#DB10.DBX60.0 BYTE 32,
              RD_1 := P#DB1002.DBX60.0 BYTE 32,
              ENO => #_w2);
   IF #_w2 THEN
       #PUT_SKV_2(REQ := "pulse_1s",   // PUT
                  ID := W#16#101,
                  ADDR_1 := P#DB10.DBX0.0 BYTE 60,
                  SD_1 := P#DB1002.DBX0.0 BYTE 60);
   END_IF;
END_REGION

REGION Network 3: SKV 3
   RUNG wire#powerrail
      "Comm_SKV_3"()
      { S7_Templates := "[remote_type := Remote, local_type := Variant]" } #GET_SKV_3.GET(REQ := "pulse_1s", ID := W#16#102, ADDR_1 := P#DB10.DBX60.0 BYTE 32, ADDR_2 :=, ADDR_3 :=, ADDR_4 :=, RD_1 := P#DB1003.DBX60.0 BYTE 32, RD_2 :=, RD_3 :=, RD_4 :=, NDR =>, ERROR =>, STATUS =>)
      { S7_Templates := "[remote_type := Remote, local_type := Variant]" } #PUT_SKV_3.PUT(REQ := "pulse_1s", ID := W#16#102, ADDR_1 := P#DB10.DBX0.0 BYTE 60, ADDR_2 :=, ADDR_3 :=, ADDR_4 :=, SD_1 := P#DB1003.DBX0.0 BYTE 60, SD_2 :=, SD_3 :=, SD_4 :=, DONE =>, ERROR =>, STATUS =>)
   END_RUNG
   // the same network as SCL:
   "Comm_SKV_3"(ENO => #_w1);   // "Comm_SKV"
   #GET_SKV_3(EN := #_w1,   // GET
              REQ := "pulse_1s",
              ID := W#16#102,
              ADDR_1 := P#DB10.DBX60.0 BYTE 32,
              RD_1 := P#DB1003.DBX60.0 BYTE 32,
              ENO => #_w2);
   IF #_w2 THEN
       #PUT_SKV_3(REQ := "pulse_1s",   // PUT
                  ID := W#16#102,
                  ADDR_1 := P#DB10.DBX0.0 BYTE 60,
                  SD_1 := P#DB1003.DBX0.0 BYTE 60);
   END_IF;
END_REGION

REGION Network 4: SKV 4
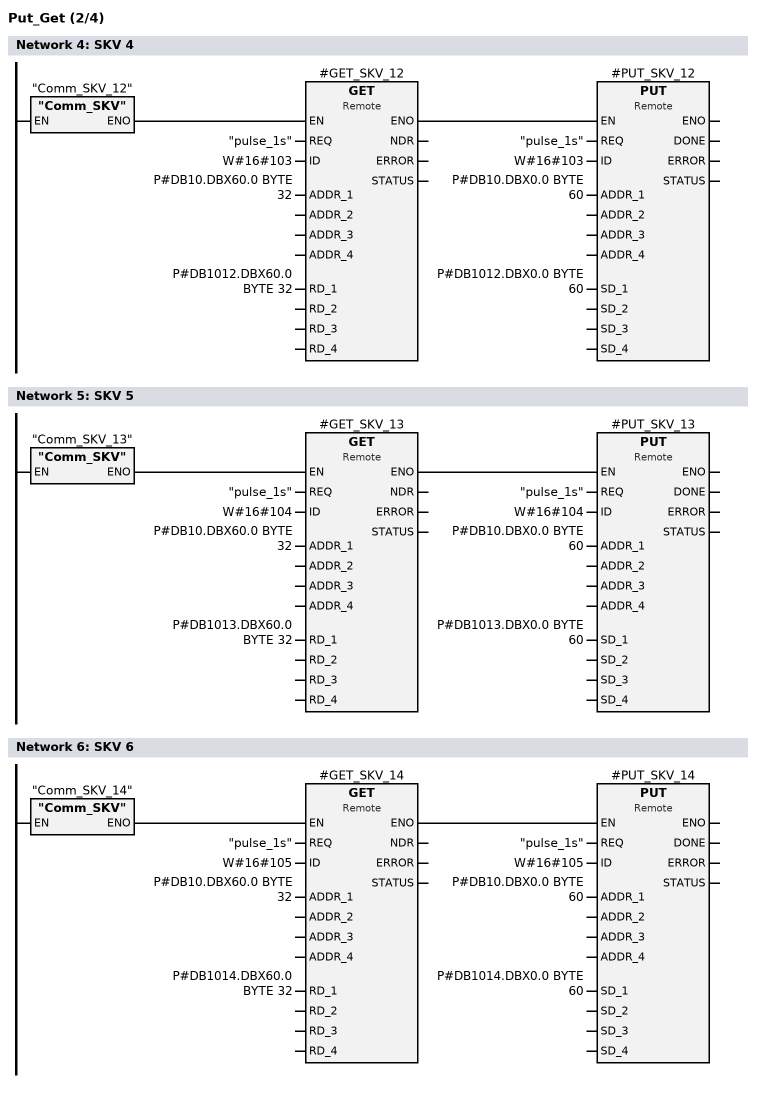
   RUNG wire#powerrail
      "Comm_SKV_12"()
      { S7_Templates := "[remote_type := Remote, local_type := Variant]" } #GET_SKV_12.GET(REQ := "pulse_1s", ID := W#16#103, ADDR_1 := P#DB10.DBX60.0 BYTE 32, ADDR_2 :=, ADDR_3 :=, ADDR_4 :=, RD_1 := P#DB1012.DBX60.0 BYTE 32, RD_2 :=, RD_3 :=, RD_4 :=, NDR =>, ERROR =>, STATUS =>)
      { S7_Templates := "[remote_type := Remote, local_type := Variant]" } #PUT_SKV_12.PUT(REQ := "pulse_1s", ID := W#16#103, ADDR_1 := P#DB10.DBX0.0 BYTE 60, ADDR_2 :=, ADDR_3 :=, ADDR_4 :=, SD_1 := P#DB1012.DBX0.0 BYTE 60, SD_2 :=, SD_3 :=, SD_4 :=, DONE =>, ERROR =>, STATUS =>)
   END_RUNG
   // the same network as SCL:
   "Comm_SKV_12"(ENO => #_w1);   // "Comm_SKV"
   #GET_SKV_12(EN := #_w1,   // GET
               REQ := "pulse_1s",
               ID := W#16#103,
               ADDR_1 := P#DB10.DBX60.0 BYTE 32,
               RD_1 := P#DB1012.DBX60.0 BYTE 32,
               ENO => #_w2);
   IF #_w2 THEN
       #PUT_SKV_12(REQ := "pulse_1s",   // PUT
                   ID := W#16#103,
                   ADDR_1 := P#DB10.DBX0.0 BYTE 60,
                   SD_1 := P#DB1012.DBX0.0 BYTE 60);
   END_IF;
END_REGION

REGION Network 5: SKV 5
   RUNG wire#powerrail
      "Comm_SKV_13"()
      { S7_Templates := "[remote_type := Remote, local_type := Variant]" } #GET_SKV_13.GET(REQ := "pulse_1s", ID := W#16#104, ADDR_1 := P#DB10.DBX60.0 BYTE 32, ADDR_2 :=, ADDR_3 :=, ADDR_4 :=, RD_1 := P#DB1013.DBX60.0 BYTE 32, RD_2 :=, RD_3 :=, RD_4 :=, NDR =>, ERROR =>, STATUS =>)
      { S7_Templates := "[remote_type := Remote, local_type := Variant]" } #PUT_SKV_13.PUT(REQ := "pulse_1s", ID := W#16#104, ADDR_1 := P#DB10.DBX0.0 BYTE 60, ADDR_2 :=, ADDR_3 :=, ADDR_4 :=, SD_1 := P#DB1013.DBX0.0 BYTE 60, SD_2 :=, SD_3 :=, SD_4 :=, DONE =>, ERROR =>, STATUS =>)
   END_RUNG
   // the same network as SCL:
   "Comm_SKV_13"(ENO => #_w1);   // "Comm_SKV"
   #GET_SKV_13(EN := #_w1,   // GET
               REQ := "pulse_1s",
               ID := W#16#104,
               ADDR_1 := P#DB10.DBX60.0 BYTE 32,
               RD_1 := P#DB1013.DBX60.0 BYTE 32,
               ENO => #_w2);
   IF #_w2 THEN
       #PUT_SKV_13(REQ := "pulse_1s",   // PUT
                   ID := W#16#104,
                   ADDR_1 := P#DB10.DBX0.0 BYTE 60,
                   SD_1 := P#DB1013.DBX0.0 BYTE 60);
   END_IF;
END_REGION

REGION Network 6: SKV 6
   RUNG wire#powerrail
      "Comm_SKV_14"()
      { S7_Templates := "[remote_type := Remote, local_type := Variant]" } #GET_SKV_14.GET(REQ := "pulse_1s", ID := W#16#105, ADDR_1 := P#DB10.DBX60.0 BYTE 32, ADDR_2 :=, ADDR_3 :=, ADDR_4 :=, RD_1 := P#DB1014.DBX60.0 BYTE 32, RD_2 :=, RD_3 :=, RD_4 :=, NDR =>, ERROR =>, STATUS =>)
      { S7_Templates := "[remote_type := Remote, local_type := Variant]" } #PUT_SKV_14.PUT(REQ := "pulse_1s", ID := W#16#105, ADDR_1 := P#DB10.DBX0.0 BYTE 60, ADDR_2 :=, ADDR_3 :=, ADDR_4 :=, SD_1 := P#DB1014.DBX0.0 BYTE 60, SD_2 :=, SD_3 :=, SD_4 :=, DONE =>, ERROR =>, STATUS =>)
   END_RUNG
   // the same network as SCL:
   "Comm_SKV_14"(ENO => #_w1);   // "Comm_SKV"
   #GET_SKV_14(EN := #_w1,   // GET
               REQ := "pulse_1s",
               ID := W#16#105,
               ADDR_1 := P#DB10.DBX60.0 BYTE 32,
               RD_1 := P#DB1014.DBX60.0 BYTE 32,
               ENO => #_w2);
   IF #_w2 THEN
       #PUT_SKV_14(REQ := "pulse_1s",   // PUT
                   ID := W#16#105,
                   ADDR_1 := P#DB10.DBX0.0 BYTE 60,
                   SD_1 := P#DB1014.DBX0.0 BYTE 60);
   END_IF;
END_REGION

REGION Network 7: SKV 7
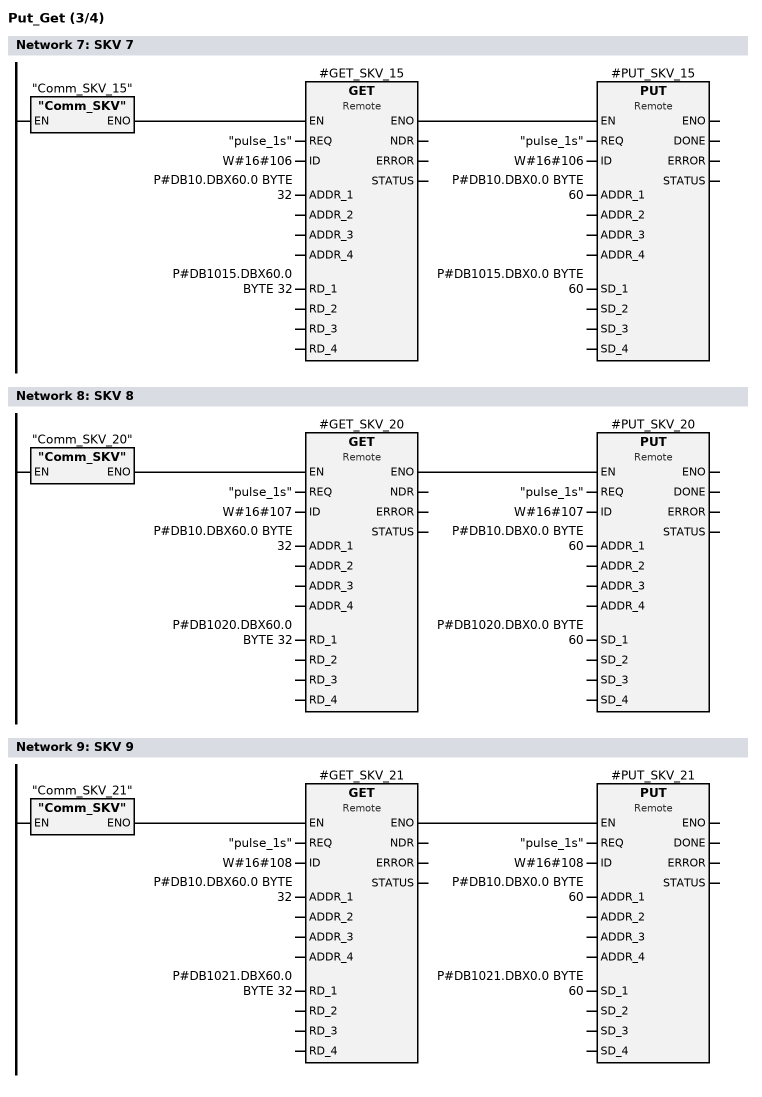
   RUNG wire#powerrail
      "Comm_SKV_15"()
      { S7_Templates := "[remote_type := Remote, local_type := Variant]" } #GET_SKV_15.GET(REQ := "pulse_1s", ID := W#16#106, ADDR_1 := P#DB10.DBX60.0 BYTE 32, ADDR_2 :=, ADDR_3 :=, ADDR_4 :=, RD_1 := P#DB1015.DBX60.0 BYTE 32, RD_2 :=, RD_3 :=, RD_4 :=, NDR =>, ERROR =>, STATUS =>)
      { S7_Templates := "[remote_type := Remote, local_type := Variant]" } #PUT_SKV_15.PUT(REQ := "pulse_1s", ID := W#16#106, ADDR_1 := P#DB10.DBX0.0 BYTE 60, ADDR_2 :=, ADDR_3 :=, ADDR_4 :=, SD_1 := P#DB1015.DBX0.0 BYTE 60, SD_2 :=, SD_3 :=, SD_4 :=, DONE =>, ERROR =>, STATUS =>)
   END_RUNG
   // the same network as SCL:
   "Comm_SKV_15"(ENO => #_w1);   // "Comm_SKV"
   #GET_SKV_15(EN := #_w1,   // GET
               REQ := "pulse_1s",
               ID := W#16#106,
               ADDR_1 := P#DB10.DBX60.0 BYTE 32,
               RD_1 := P#DB1015.DBX60.0 BYTE 32,
               ENO => #_w2);
   IF #_w2 THEN
       #PUT_SKV_15(REQ := "pulse_1s",   // PUT
                   ID := W#16#106,
                   ADDR_1 := P#DB10.DBX0.0 BYTE 60,
                   SD_1 := P#DB1015.DBX0.0 BYTE 60);
   END_IF;
END_REGION

REGION Network 8: SKV 8
   RUNG wire#powerrail
      "Comm_SKV_20"()
      { S7_Templates := "[remote_type := Remote, local_type := Variant]" } #GET_SKV_20.GET(REQ := "pulse_1s", ID := W#16#107, ADDR_1 := P#DB10.DBX60.0 BYTE 32, ADDR_2 :=, ADDR_3 :=, ADDR_4 :=, RD_1 := P#DB1020.DBX60.0 BYTE 32, RD_2 :=, RD_3 :=, RD_4 :=, NDR =>, ERROR =>, STATUS =>)
      { S7_Templates := "[remote_type := Remote, local_type := Variant]" } #PUT_SKV_20.PUT(REQ := "pulse_1s", ID := W#16#107, ADDR_1 := P#DB10.DBX0.0 BYTE 60, ADDR_2 :=, ADDR_3 :=, ADDR_4 :=, SD_1 := P#DB1020.DBX0.0 BYTE 60, SD_2 :=, SD_3 :=, SD_4 :=, DONE =>, ERROR =>, STATUS =>)
   END_RUNG
   // the same network as SCL:
   "Comm_SKV_20"(ENO => #_w1);   // "Comm_SKV"
   #GET_SKV_20(EN := #_w1,   // GET
               REQ := "pulse_1s",
               ID := W#16#107,
               ADDR_1 := P#DB10.DBX60.0 BYTE 32,
               RD_1 := P#DB1020.DBX60.0 BYTE 32,
               ENO => #_w2);
   IF #_w2 THEN
       #PUT_SKV_20(REQ := "pulse_1s",   // PUT
                   ID := W#16#107,
                   ADDR_1 := P#DB10.DBX0.0 BYTE 60,
                   SD_1 := P#DB1020.DBX0.0 BYTE 60);
   END_IF;
END_REGION

REGION Network 9: SKV 9
   RUNG wire#powerrail
      "Comm_SKV_21"()
      { S7_Templates := "[remote_type := Remote, local_type := Variant]" } #GET_SKV_21.GET(REQ := "pulse_1s", ID := W#16#108, ADDR_1 := P#DB10.DBX60.0 BYTE 32, ADDR_2 :=, ADDR_3 :=, ADDR_4 :=, RD_1 := P#DB1021.DBX60.0 BYTE 32, RD_2 :=, RD_3 :=, RD_4 :=, NDR =>, ERROR =>, STATUS =>)
      { S7_Templates := "[remote_type := Remote, local_type := Variant]" } #PUT_SKV_21.PUT(REQ := "pulse_1s", ID := W#16#108, ADDR_1 := P#DB10.DBX0.0 BYTE 60, ADDR_2 :=, ADDR_3 :=, ADDR_4 :=, SD_1 := P#DB1021.DBX0.0 BYTE 60, SD_2 :=, SD_3 :=, SD_4 :=, DONE =>, ERROR =>, STATUS =>)
   END_RUNG
   // the same network as SCL:
   "Comm_SKV_21"(ENO => #_w1);   // "Comm_SKV"
   #GET_SKV_21(EN := #_w1,   // GET
               REQ := "pulse_1s",
               ID := W#16#108,
               ADDR_1 := P#DB10.DBX60.0 BYTE 32,
               RD_1 := P#DB1021.DBX60.0 BYTE 32,
               ENO => #_w2);
   IF #_w2 THEN
       #PUT_SKV_21(REQ := "pulse_1s",   // PUT
                   ID := W#16#108,
                   ADDR_1 := P#DB10.DBX0.0 BYTE 60,
                   SD_1 := P#DB1021.DBX0.0 BYTE 60);
   END_IF;
END_REGION

REGION Network 10: SKV 10
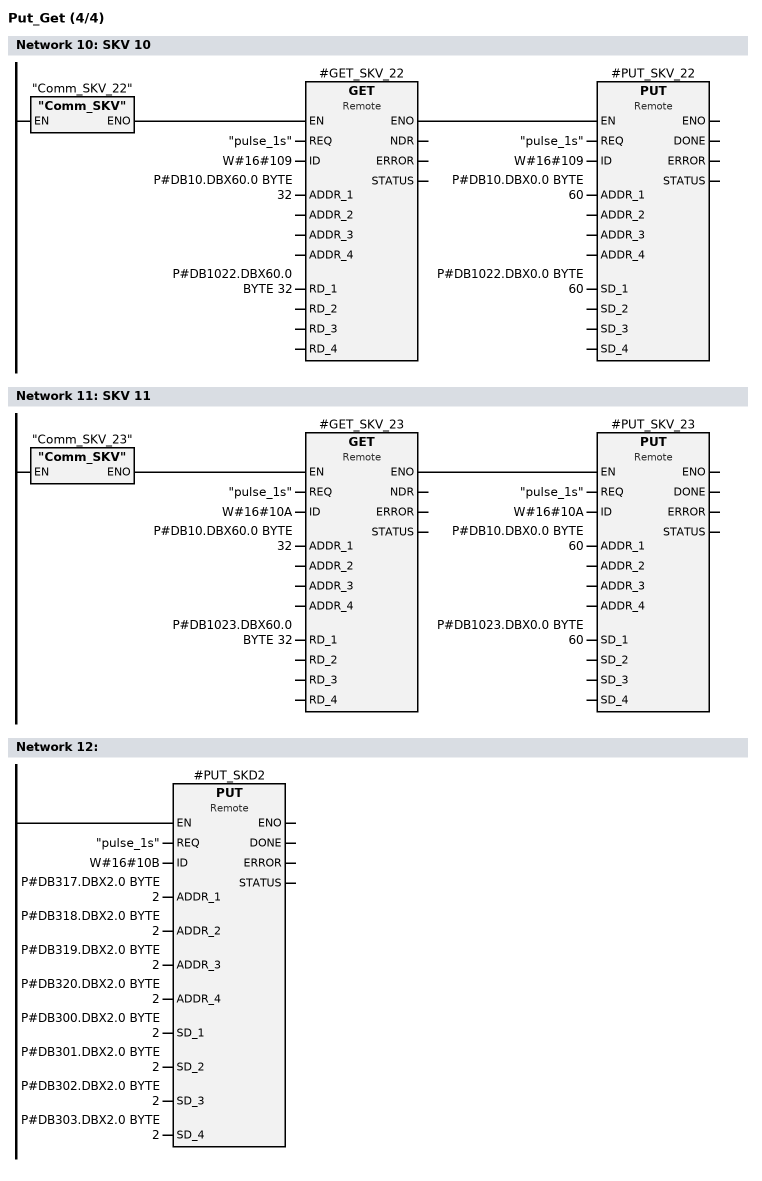
   RUNG wire#powerrail
      "Comm_SKV_22"()
      { S7_Templates := "[remote_type := Remote, local_type := Variant]" } #GET_SKV_22.GET(REQ := "pulse_1s", ID := W#16#109, ADDR_1 := P#DB10.DBX60.0 BYTE 32, ADDR_2 :=, ADDR_3 :=, ADDR_4 :=, RD_1 := P#DB1022.DBX60.0 BYTE 32, RD_2 :=, RD_3 :=, RD_4 :=, NDR =>, ERROR =>, STATUS =>)
      { S7_Templates := "[remote_type := Remote, local_type := Variant]" } #PUT_SKV_22.PUT(REQ := "pulse_1s", ID := W#16#109, ADDR_1 := P#DB10.DBX0.0 BYTE 60, ADDR_2 :=, ADDR_3 :=, ADDR_4 :=, SD_1 := P#DB1022.DBX0.0 BYTE 60, SD_2 :=, SD_3 :=, SD_4 :=, DONE =>, ERROR =>, STATUS =>)
   END_RUNG
   // the same network as SCL:
   "Comm_SKV_22"(ENO => #_w1);   // "Comm_SKV"
   #GET_SKV_22(EN := #_w1,   // GET
               REQ := "pulse_1s",
               ID := W#16#109,
               ADDR_1 := P#DB10.DBX60.0 BYTE 32,
               RD_1 := P#DB1022.DBX60.0 BYTE 32,
               ENO => #_w2);
   IF #_w2 THEN
       #PUT_SKV_22(REQ := "pulse_1s",   // PUT
                   ID := W#16#109,
                   ADDR_1 := P#DB10.DBX0.0 BYTE 60,
                   SD_1 := P#DB1022.DBX0.0 BYTE 60);
   END_IF;
END_REGION

REGION Network 11: SKV 11
   RUNG wire#powerrail
      "Comm_SKV_23"()
      { S7_Templates := "[remote_type := Remote, local_type := Variant]" } #GET_SKV_23.GET(REQ := "pulse_1s", ID := W#16#10A, ADDR_1 := P#DB10.DBX60.0 BYTE 32, ADDR_2 :=, ADDR_3 :=, ADDR_4 :=, RD_1 := P#DB1023.DBX60.0 BYTE 32, RD_2 :=, RD_3 :=, RD_4 :=, NDR =>, ERROR =>, STATUS =>)
      { S7_Templates := "[remote_type := Remote, local_type := Variant]" } #PUT_SKV_23.PUT(REQ := "pulse_1s", ID := W#16#10A, ADDR_1 := P#DB10.DBX0.0 BYTE 60, ADDR_2 :=, ADDR_3 :=, ADDR_4 :=, SD_1 := P#DB1023.DBX0.0 BYTE 60, SD_2 :=, SD_3 :=, SD_4 :=, DONE =>, ERROR =>, STATUS =>)
   END_RUNG
   // the same network as SCL:
   "Comm_SKV_23"(ENO => #_w1);   // "Comm_SKV"
   #GET_SKV_23(EN := #_w1,   // GET
               REQ := "pulse_1s",
               ID := W#16#10A,
               ADDR_1 := P#DB10.DBX60.0 BYTE 32,
               RD_1 := P#DB1023.DBX60.0 BYTE 32,
               ENO => #_w2);
   IF #_w2 THEN
       #PUT_SKV_23(REQ := "pulse_1s",   // PUT
                   ID := W#16#10A,
                   ADDR_1 := P#DB10.DBX0.0 BYTE 60,
                   SD_1 := P#DB1023.DBX0.0 BYTE 60);
   END_IF;
END_REGION

REGION Network 12
   RUNG wire#powerrail
      { S7_Templates := "[remote_type := Remote, local_type := Variant]" } #PUT_SKD2.PUT(REQ := "pulse_1s", ID := W#16#10B, ADDR_1 := P#DB317.DBX2.0 BYTE 2, ADDR_2 := P#DB318.DBX2.0 BYTE 2, ADDR_3 := P#DB319.DBX2.0 BYTE 2, ADDR_4 := P#DB320.DBX2.0 BYTE 2, SD_1 := P#DB300.DBX2.0 BYTE 2, SD_2 := P#DB301.DBX2.0 BYTE 2, SD_3 := P#DB302.DBX2.0 BYTE 2, SD_4 := P#DB303.DBX2.0 BYTE 2, DONE =>, ERROR =>, STATUS =>)
   END_RUNG
   // the same network as SCL:
   #PUT_SKD2(REQ := "pulse_1s",   // PUT
             ID := W#16#10B,
             ADDR_1 := P#DB317.DBX2.0 BYTE 2,
             ADDR_2 := P#DB318.DBX2.0 BYTE 2,
             ADDR_3 := P#DB319.DBX2.0 BYTE 2,
             ADDR_4 := P#DB320.DBX2.0 BYTE 2,
             SD_1 := P#DB300.DBX2.0 BYTE 2,
             SD_2 := P#DB301.DBX2.0 BYTE 2,
             SD_3 := P#DB302.DBX2.0 BYTE 2,
             SD_4 := P#DB303.DBX2.0 BYTE 2);
END_REGION
END_FUNCTION_BLOCK

FUNCTION_BLOCK "Comm_SKV"
{ S7_Optimized_Access := 'FALSE' }
VERSION : 0.1
   VAR 
      To_SKV : Struct
         watchdog : Int;
         LE_1 : Int;
         LE_2 : Int;
         LE_3 : Int;
         LE_4 : Int;
         SP_FE : Int;
         SP_M : Int;
         CMD : Struct
            REQ : Bool;
            Reset : Bool;
            Hand : Bool;
            Start_M : Bool;
         END_STRUCT;
         Valves : Struct
            ID : Int;
            Local : Array[0..15] of Bool;
            Mode : Array[1..10] of Int;
            Status : Array[1..10] of Int;
         END_STRUCT;
      END_STRUCT;
      From_SKV : Struct
         watchdog : Int;
         LE_SKV : Int;
         res_h : DInt;
         LE : Int;
         TE : Int;
         PE_1 : Int;
         PE_2 : Int;
         PE_3 : Int;
         PE_4 : Int;
         FE : Int;
         C : Int;
         Status : Int;
         STATE : Struct
            Ready : Bool;
            Local : Bool;
            Warning : Bool;
            Alarm : Bool;
            LS : Bool;
            Lock : Bool;
         END_STRUCT;
         Valves : Struct
            ID : Int;
            REQ : Array[0..15] of Bool;
         END_STRUCT;
      END_STRUCT;
      watchdog_control : Int;
      Alarm : Struct
         Link : Bool;
      END_STRUCT;
      ID : Int;
      SP_M : Real;
      SP_FE : Real;
      LE : Real;
      PE_1 : Real;
      PE_2 : Real;
      PE_3 : Real;
      PE_4 : Real;
      FE : Real;
      TE : Real;
      C : Real;
      Route : Bool;
      "Name" : Array[0..10] of String[5];
      Clock { S7_SetPoint := 'False'} : Array[0..10] of "Time_S";
   END_VAR

   VAR_TEMP 
      x : Int;
   END_VAR


BEGIN
	//Отправка данных в СКВ
	    //контроль связи
	    IF #watchdog_control = #From_SKV.watchdog THEN
	        #Clock[0].Start := TRUE;
	        IF #Clock[0]."Exit" THEN
	            #Alarm.Link := TRUE; //нет связи с ЩКД1
	        ELSE
	            #Alarm.Link := FALSE;
	        END_IF;
	    ELSE
	        #Clock[0].Start := FALSE;
	    END_IF;
	    
	    //уровни в РВ
	    #To_SKV.LE_1 := REAL_TO_INT("LE_105".Result * 10.0);
	    #To_SKV.LE_2 := REAL_TO_INT("LE_106".Result * 10.0);
	    #To_SKV.LE_3 := REAL_TO_INT("LE_107".Result * 10.0);
	    #To_SKV.LE_4 := REAL_TO_INT("LE_108".Result * 10.0);
	    
	    //управление насосом
	    #To_SKV.SP_M := REAL_TO_INT(#SP_M * 10.0);
	    
	    //сброс аварий
	    IF #To_SKV.CMD.Reset THEN
	        #Clock[1].Start := TRUE;
	        IF #Clock[1]."Exit" THEN
	            #To_SKV.CMD.Reset := FALSE;
	            #Clock[1].Start := FALSE;
	        END_IF;
	    END_IF;
	    
	    //статусы задвижек
	    CASE #ID OF
	        0:  //КП не выбрано
	            FOR #x := 1 TO 10 DO
	                #To_SKV.Valves.Status[#x] := 0;
	            END_FOR;
	        1:  //КП 2.1
	            FOR #x := 1 TO 10 DO
	                #To_SKV.Valves.Status[#x] := "KP_2_1_DB".KP[#x].Status;
	            END_FOR;
	        2:  //КП 2.1
	            FOR #x := 1 TO 10 DO
	                #To_SKV.Valves.Status[#x] := "KP_2_2_DB".KP[#x].Status;
	            END_FOR;
	        3:  //КП 2.3
	            FOR #x := 1 TO 10 DO
	                #To_SKV.Valves.Status[#x] := "KP_2_3_DB".KP[#x].Status;
	            END_FOR;
	        4:  //КП 2.4
	            FOR #x := 1 TO 10 DO
	                #To_SKV.Valves.Status[#x] := "KP_2_4_DB".KP[#x].Status;
	            END_FOR;
	        5:  //КП 2.5
	            FOR #x := 1 TO 10 DO
	                #To_SKV.Valves.Status[#x] := "KP_2_5_DB".KP[#x].Status;
	            END_FOR;
	        6:  //КП 2.6
	            FOR #x := 1 TO 10 DO
	                #To_SKV.Valves.Status[#x] := "KP_2_6_DB".KP[#x].Status;
	            END_FOR;
	        7:  //КП 2.7
	            FOR #x := 1 TO 10 DO
	                #To_SKV.Valves.Status[#x] := "KP_2_7_DB".KP[#x].Status;
	            END_FOR;
	        8:  //КП 2.8
	            FOR #x := 1 TO 10 DO
	                #To_SKV.Valves.Status[#x] := "KP_2_8_DB".KP[#x].Status;
	            END_FOR;
	        9:  //КП 2.9
	            FOR #x := 1 TO 10 DO
	                #To_SKV.Valves.Status[#x] := "KP_2_9_DB".KP[#x].Status;
	            END_FOR;
	        10:  //КП 2.10
	            FOR #x := 1 TO 10 DO
	                #To_SKV.Valves.Status[#x] := "KP_2_10_DB".KP[#x].Status;
	            END_FOR;
	    END_CASE;
	
	    
	//Получение данных от СКВ
	    //контроль связи
	    IF "pulse_1s" THEN
	        #To_SKV.watchdog := #To_SKV.watchdog + 1;
	        IF #To_SKV.watchdog > 10000 THEN
	            #To_SKV.watchdog := 0;
	        END_IF;
	    END_IF;
	    
	    #ID := #From_SKV.Valves.ID;
	
	    //давление в КП
	    #PE_1 := INT_TO_REAL(#From_SKV.PE_1) / 10;
	    #PE_2 := INT_TO_REAL(#From_SKV.PE_2) / 10;
	    #PE_3 := INT_TO_REAL(#From_SKV.PE_3) / 10;
	    #PE_4 := INT_TO_REAL(#From_SKV.PE_4) / 10;
	    
	    //прочие датчики
	    #LE := INT_TO_REAL(#From_SKV.LE) / 10;
	    #TE := INT_TO_REAL(#From_SKV.TE) / 10;
	    #FE := INT_TO_REAL(#From_SKV.FE) / 10;
	    #C := INT_TO_REAL(#From_SKV.C) / 10;
	    
	    
	//вызов таймеров на исполнение
	FOR #x := 0 TO 10 BY 1 DO
	    #Clock[#x]();
	END_FOR;
END_FUNCTION_BLOCK

FUNCTION "FC_DRV_End" : Void   // FC101, LAD
{ S7_Optimized_Access := 'FALSE' }
VERSION : 0.1
// stored: AutoNumber false, IsIECCheckEnabled false, SetENOAutomatically false, UDAEnableTagReadback false
   VAR_TEMP
      ev : Bool;
   END_VAR
   VAR_TEMP   // added for the SCL form of the ladder/FBD networks
      _w1 : Bool;
      _w2 : Bool;
      _w3 : Bool;
      _w4 : Bool;
      _w5 : Bool;
      _w6 : Bool;
      _w7 : Bool;
      _w8 : Bool;
   END_VAR
BEGIN

REGION Network 1: Одно из устройств нижнего уровня в ручном режиме
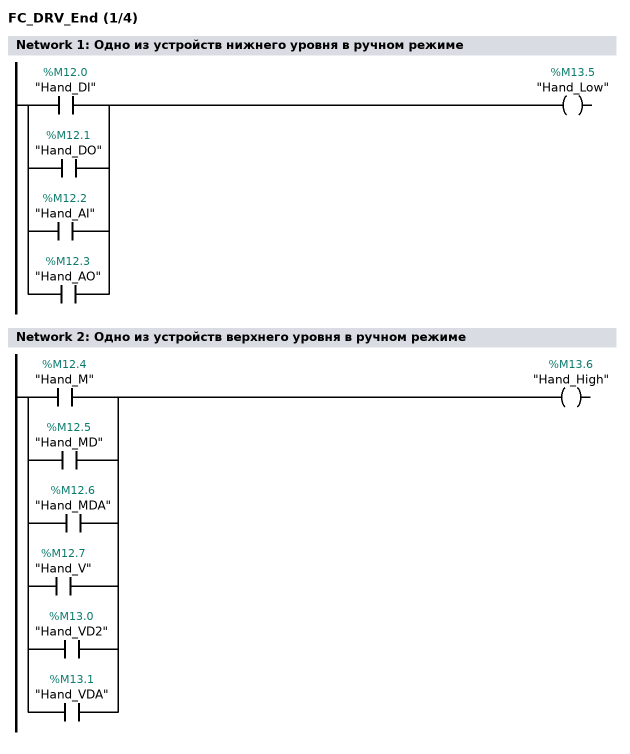
   RUNG wire#powerrail
      Contact( "Hand_DI" )
      wire#w1
      Coil( "Hand_Low" )
   END_RUNG
   RUNG wire#powerrail
      Contact( "Hand_DO" )
   END_RUNG wire#w1
   RUNG wire#powerrail
      Contact( "Hand_AI" )
   END_RUNG wire#w1
   RUNG wire#powerrail
      Contact( "Hand_AO" )
   END_RUNG wire#w1
   // the same network as SCL:
   "Hand_Low" := "Hand_DI" OR "Hand_DO" OR "Hand_AI" OR "Hand_AO";
END_REGION

REGION Network 2: Одно из устройств верхнего уровня в ручном режиме
   RUNG wire#powerrail
      Contact( "Hand_M" )
      wire#w1
      Coil( "Hand_High" )
   END_RUNG
   RUNG wire#powerrail
      Contact( "Hand_MD" )
   END_RUNG wire#w1
   RUNG wire#powerrail
      Contact( "Hand_MDA" )
   END_RUNG wire#w1
   RUNG wire#powerrail
      Contact( "Hand_V" )
   END_RUNG wire#w1
   RUNG wire#powerrail
      Contact( "Hand_VD2" )
   END_RUNG wire#w1
   RUNG wire#powerrail
      Contact( "Hand_VDA" )
   END_RUNG wire#w1
   // the same network as SCL:
   "Hand_High" := "Hand_M" OR "Hand_MD" OR "Hand_MDA" OR "Hand_V" OR "Hand_VD2" OR "Hand_VDA";
END_REGION

REGION Network 3: Сбор и сброс статусов ручного режима
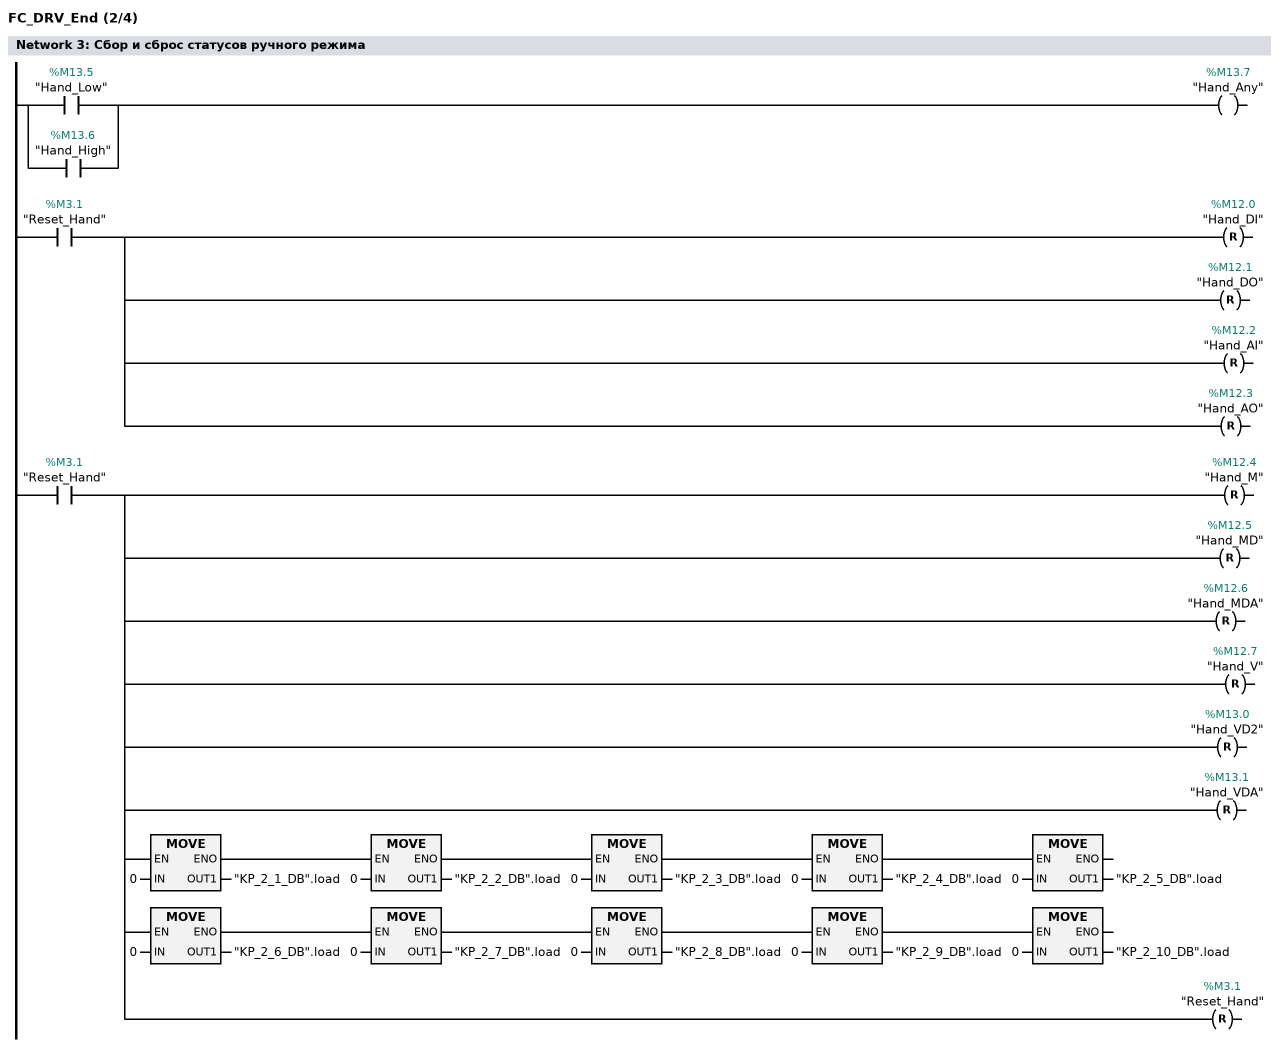
   RUNG wire#powerrail
      Contact( "Hand_Low" )
      wire#w1
      Coil( "Hand_Any" )
   END_RUNG
   RUNG wire#powerrail
      Contact( "Hand_High" )
   END_RUNG wire#w1
   RUNG wire#powerrail
      Contact( "Reset_Hand" )
      wire#w2
      R_Coil( "Hand_DI" )
   END_RUNG
   RUNG wire#w2
      R_Coil( "Hand_DO" )
   END_RUNG
   RUNG wire#w2
      R_Coil( "Hand_AI" )
   END_RUNG
   RUNG wire#w2
      R_Coil( "Hand_AO" )
   END_RUNG
   RUNG wire#powerrail
      Contact( "Reset_Hand" )
      wire#w3
      R_Coil( "Hand_M" )
   END_RUNG
   RUNG wire#w3
      R_Coil( "Hand_MD" )
   END_RUNG
   RUNG wire#w3
      R_Coil( "Hand_MDA" )
   END_RUNG
   RUNG wire#w3
      R_Coil( "Hand_V" )
   END_RUNG
   RUNG wire#w3
      R_Coil( "Hand_VD2" )
   END_RUNG
   RUNG wire#w3
      R_Coil( "Hand_VDA" )
   END_RUNG
   RUNG wire#w3
      Move(in := 0, out1 => "KP_2_1_DB".load)
      Move(in := 0, out1 => "KP_2_2_DB".load)
      Move(in := 0, out1 => "KP_2_3_DB".load)
      Move(in := 0, out1 => "KP_2_4_DB".load)
      Move(in := 0, out1 => "KP_2_5_DB".load)
   END_RUNG
   RUNG wire#w3
      Move(in := 0, out1 => "KP_2_6_DB".load)
      Move(in := 0, out1 => "KP_2_7_DB".load)
      Move(in := 0, out1 => "KP_2_8_DB".load)
      Move(in := 0, out1 => "KP_2_9_DB".load)
      Move(in := 0, out1 => "KP_2_10_DB".load)
   END_RUNG
   RUNG wire#w3
      R_Coil( "Reset_Hand" )
   END_RUNG
   // the same network as SCL:
   "Hand_Any" := "Hand_Low" OR "Hand_High";
   IF "Reset_Hand" THEN
       "Hand_DI" := FALSE;
       "Hand_DO" := FALSE;
       "Hand_AI" := FALSE;
       "Hand_AO" := FALSE;
       "Hand_M" := FALSE;
       "Hand_MD" := FALSE;
       "Hand_MDA" := FALSE;
       "Hand_V" := FALSE;
       "Hand_VD2" := FALSE;
       "Hand_VDA" := FALSE;
       "KP_2_1_DB".load := 0;
       "KP_2_2_DB".load := 0;
       "KP_2_3_DB".load := 0;
       "KP_2_4_DB".load := 0;
       "KP_2_5_DB".load := 0;
       "KP_2_6_DB".load := 0;
       "KP_2_7_DB".load := 0;
       "KP_2_8_DB".load := 0;
       "KP_2_9_DB".load := 0;
       "KP_2_10_DB".load := 0;
       "Reset_Hand" := FALSE;
   END_IF;
END_REGION

REGION Network 4
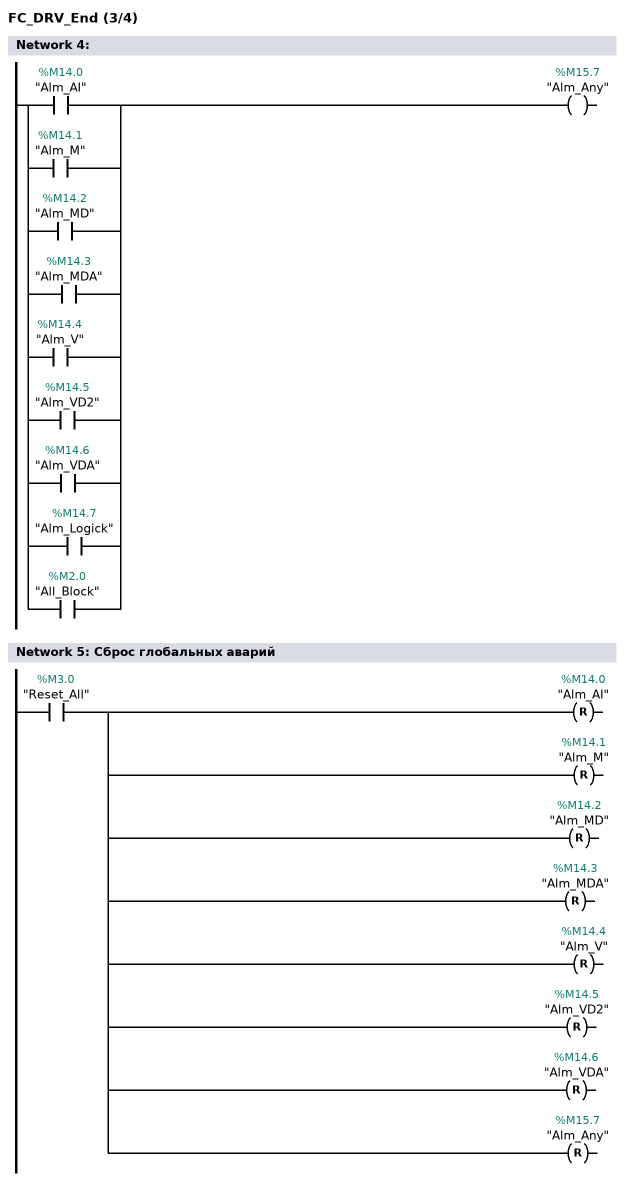
   RUNG wire#powerrail
      Contact( "Alm_AI" )
      wire#w1
      Coil( "Alm_Any" )
   END_RUNG
   RUNG wire#powerrail
      Contact( "Alm_M" )
   END_RUNG wire#w1
   RUNG wire#powerrail
      Contact( "Alm_MD" )
   END_RUNG wire#w1
   RUNG wire#powerrail
      Contact( "Alm_MDA" )
   END_RUNG wire#w1
   RUNG wire#powerrail
      Contact( "Alm_V" )
   END_RUNG wire#w1
   RUNG wire#powerrail
      Contact( "Alm_VD2" )
   END_RUNG wire#w1
   RUNG wire#powerrail
      Contact( "Alm_VDA" )
   END_RUNG wire#w1
   RUNG wire#powerrail
      Contact( "Alm_Logick" )
   END_RUNG wire#w1
   RUNG wire#powerrail
      Contact( "All_Block" )
   END_RUNG wire#w1
   // the same network as SCL:
   "Alm_Any" := "Alm_AI" OR "Alm_M" OR "Alm_MD" OR "Alm_MDA" OR "Alm_V" OR "Alm_VD2" OR "Alm_VDA" OR "Alm_Logick" OR "All_Block";
END_REGION

REGION Network 5: Сброс глобальных аварий
   RUNG wire#powerrail
      Contact( "Reset_All" )
      wire#w1
      R_Coil( "Alm_AI" )
   END_RUNG
   RUNG wire#w1
      R_Coil( "Alm_M" )
   END_RUNG
   RUNG wire#w1
      R_Coil( "Alm_MD" )
   END_RUNG
   RUNG wire#w1
      R_Coil( "Alm_MDA" )
   END_RUNG
   RUNG wire#w1
      R_Coil( "Alm_V" )
   END_RUNG
   RUNG wire#w1
      R_Coil( "Alm_VD2" )
   END_RUNG
   RUNG wire#w1
      R_Coil( "Alm_VDA" )
   END_RUNG
   RUNG wire#w1
      R_Coil( "Alm_Any" )
   END_RUNG
   // the same network as SCL:
   IF "Reset_All" THEN
       "Alm_AI" := FALSE;
       "Alm_M" := FALSE;
       "Alm_MD" := FALSE;
       "Alm_MDA" := FALSE;
       "Alm_V" := FALSE;
       "Alm_VD2" := FALSE;
       "Alm_VDA" := FALSE;
       "Alm_Any" := FALSE;
   END_IF;
END_REGION

REGION Network 6: Основные события
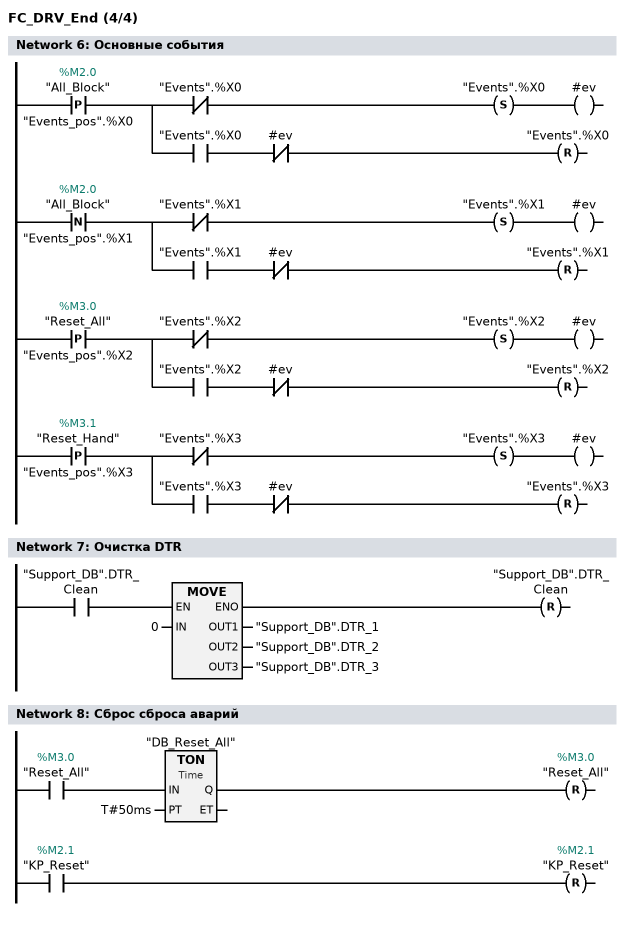
   RUNG wire#powerrail
      P_Contact(operand := "All_Block", bit := "Events_pos".%X0)
      wire#w1
      I_Contact( "Events".%X0 )
      S_Coil( "Events".%X0 )
      Coil( #ev )
   END_RUNG
   RUNG wire#w1
      Contact( "Events".%X0 )
      I_Contact( #ev )
      R_Coil( "Events".%X0 )
   END_RUNG
   RUNG wire#powerrail
      N_Contact(operand := "All_Block", bit := "Events_pos".%X1)
      wire#w2
      I_Contact( "Events".%X1 )
      S_Coil( "Events".%X1 )
      Coil( #ev )
   END_RUNG
   RUNG wire#w2
      Contact( "Events".%X1 )
      I_Contact( #ev )
      R_Coil( "Events".%X1 )
   END_RUNG
   RUNG wire#powerrail
      P_Contact(operand := "Reset_All", bit := "Events_pos".%X2)
      wire#w3
      I_Contact( "Events".%X2 )
      S_Coil( "Events".%X2 )
      Coil( #ev )
   END_RUNG
   RUNG wire#w3
      Contact( "Events".%X2 )
      I_Contact( #ev )
      R_Coil( "Events".%X2 )
   END_RUNG
   RUNG wire#powerrail
      P_Contact(operand := "Reset_Hand", bit := "Events_pos".%X3)
      wire#w4
      I_Contact( "Events".%X3 )
      S_Coil( "Events".%X3 )
      Coil( #ev )
   END_RUNG
   RUNG wire#w4
      Contact( "Events".%X3 )
      I_Contact( #ev )
      R_Coil( "Events".%X3 )
   END_RUNG
   // the same network as SCL:
   #_w1 := "All_Block" AND NOT "Events_pos".%X0;   // rising edge of "All_Block"
   "Events_pos".%X0 := "All_Block";
   #_w2 := #_w1 AND NOT "Events".%X0;
   IF #_w2 THEN "Events".%X0 := TRUE; END_IF;
   #ev := #_w2;
   IF #_w1 AND "Events".%X0 AND NOT #ev THEN "Events".%X0 := FALSE; END_IF;
   #_w3 := NOT "All_Block" AND "Events_pos".%X1;   // falling edge of "All_Block"
   "Events_pos".%X1 := "All_Block";
   #_w4 := #_w3 AND NOT "Events".%X1;
   IF #_w4 THEN "Events".%X1 := TRUE; END_IF;
   #ev := #_w4;
   IF #_w3 AND "Events".%X1 AND NOT #ev THEN "Events".%X1 := FALSE; END_IF;
   #_w5 := "Reset_All" AND NOT "Events_pos".%X2;   // rising edge of "Reset_All"
   "Events_pos".%X2 := "Reset_All";
   #_w6 := #_w5 AND NOT "Events".%X2;
   IF #_w6 THEN "Events".%X2 := TRUE; END_IF;
   #ev := #_w6;
   IF #_w5 AND "Events".%X2 AND NOT #ev THEN "Events".%X2 := FALSE; END_IF;
   #_w7 := "Reset_Hand" AND NOT "Events_pos".%X3;   // rising edge of "Reset_Hand"
   "Events_pos".%X3 := "Reset_Hand";
   #_w8 := #_w7 AND NOT "Events".%X3;
   IF #_w8 THEN "Events".%X3 := TRUE; END_IF;
   #ev := #_w8;
   IF #_w7 AND "Events".%X3 AND NOT #ev THEN "Events".%X3 := FALSE; END_IF;
END_REGION

REGION Network 7: Очистка DTR
   RUNG wire#powerrail
      Contact( "Support_DB".DTR_Clean )
      Move(in := 0, out1 => "Support_DB".DTR_1, out2 => "Support_DB".DTR_2, out3 => "Support_DB".DTR_3)
      R_Coil( "Support_DB".DTR_Clean )
   END_RUNG
   // the same network as SCL:
   IF "Support_DB".DTR_Clean THEN
       "Support_DB".DTR_1 := 0;
       "Support_DB".DTR_2 := 0;
       "Support_DB".DTR_3 := 0;
       "Support_DB".DTR_Clean := FALSE;
   END_IF;
END_REGION

REGION Network 8: Сброс сброса аварий
   RUNG wire#powerrail
      Contact( "Reset_All" )
      { S7_Templates := "time_type := Time" } "DB_Reset_All".TON(pt := T#50ms, et =>)
      R_Coil( "Reset_All" )
   END_RUNG
   RUNG wire#powerrail
      Contact( "KP_Reset" )
      R_Coil( "KP_Reset" )
   END_RUNG
   // the same network as SCL:
   "DB_Reset_All".TON(IN := "Reset_All", PT := T#50ms);
   IF "DB_Reset_All".Q THEN "Reset_All" := FALSE; END_IF;
   IF "KP_Reset" THEN "KP_Reset" := FALSE; END_IF;
END_REGION
END_FUNCTION

ORGANIZATION_BLOCK "Cyclic interrupt"   // OB30, LAD, CyclicInterrupt
{ S7_Optimized_Access := 'TRUE' }
VERSION : 0.1
// stored: AutoNumber true, IsIECCheckEnabled false, SetENOAutomatically false
   VAR_INPUT
      Initial_Call : Bool;   // Initial call of this OB
      Event_Count : Int;   // Events discarded
   END_VAR
BEGIN

REGION Network 1
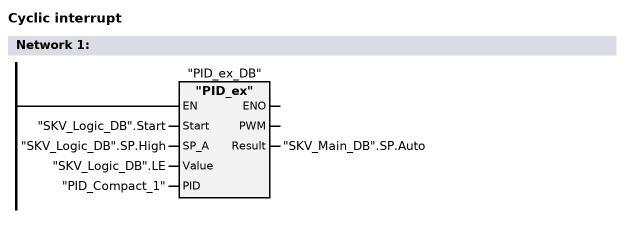
   RUNG wire#powerrail
      "PID_ex_DB"(Start := "SKV_Logic_DB".Start, SP_A := "SKV_Logic_DB".SP.High, Value := "SKV_Logic_DB".LE, PID := "PID_Compact_1", PWM =>, Result => "SKV_Main_DB".SP.Auto)
   END_RUNG
   // the same network as SCL:
   "PID_ex_DB"(Start := "SKV_Logic_DB".Start,   // "PID_ex"
               SP_A := "SKV_Logic_DB".SP.High,
               Value := "SKV_Logic_DB".LE,
               PID := "PID_Compact_1",
               Result => "SKV_Main_DB".SP.Auto);
END_REGION
END_ORGANIZATION_BLOCK

FUNCTION_BLOCK "PID_ex"   // FB99, LAD
TITLE = Обвязка ПИД-регулятора
{ S7_Optimized_Access := 'FALSE' }
VERSION : 0.1
// stored: AutoNumber false, IsIECCheckEnabled false, SetENOAutomatically false, UDAEnableTagReadback false
   VAR_INPUT
      Start : Bool;
      SP_A : Real;   // Уставка
      Value : Real;   // Показания датчика
   END_VAR
   VAR_OUTPUT
      PWM : Bool;   // ШИМ-выход ПИД-регулятора
      Result : Real;   // Управляющее воздействие
   END_VAR
   VAR_IN_OUT
      PID : PID_Compact;   // ПИД
   END_VAR
   VAR DB_SPECIFIC
      CMD : "CMD";
      SP_M : Real;
      SP : Real;
      x { S7_SetPoint := 'True'} : Real := 1.0;   // Поправка уставки и датчика
      SP_x : Real;   // Домноженная уставка
      Value_x : Real;   // Домноженный датчик
      Buffer : Real;   // Промежуточное значение
      PID_Output : Real;   // Выход ПИД-регулятора
      PID_Hand : Real;   // Ручное задание выхода ПИД-регулятора
      Sys : Struct   // Системные параметры
         Err_Ack : Bool;   // Подтверждение аварии
         Alm_SP_H : Bool;   // Авария уставки - превышение
         Alm_SP_L : Bool;   // Авария уставки - занижение
         Alm_In_H : Bool;   // Авария датчика - превышение
         Alm_In_L : Bool;   // Авария датчика - занижение
         Activate : Bool;   // Активировать ПИД
         First_Run { S7_SetPoint := 'True'} : Bool;   // Первый пуск
         Error_code : DWord;   // Код аварии
         Warning_code : DWord;   // Код предупреждения
         "Type" : Int := 1;   // Режим работы
         State : Int;   // Состояние
         Mode : Int := 3;   // Режим
      END_STRUCT;
      Settings : Struct   // Рабочие параметры
         SP_P { S7_SetPoint := 'True'} : Real := 1.5;   // Коэффициент пропорциональности
         SP_Ti { S7_SetPoint := 'True'} : Real := 150.0;   // Время интегрирования
         SP_Td { S7_SetPoint := 'True'} : Real;   // Время дифференцирования
         SP_Cycle { S7_SetPoint := 'True'} : Real := 0.2;   // Время цикла
         Max_SP { S7_SetPoint := 'True'} : Real := 500.0;   // Максимальное значение уставки
         Min_SP { S7_SetPoint := 'True'} : Real := -500.0;   // Минимальное значение уставки
         Max_in { S7_SetPoint := 'True'} : Real := 500.0;   // Максимальное значение датчика
         Min_in { S7_SetPoint := 'True'} : Real := -500.0;   // Минимальное значение датчика
         Max_out { S7_SetPoint := 'True'} : Real := 100.0;   // Максимальное значение выхода
         Min_out { S7_SetPoint := 'True'} : Real := 0.0;   // Минимальное значение выхода
         DeadBand { S7_SetPoint := 'True'} : Real := 1.0;   // Мёртвая зона
         Max : Real;   // Верняя граница мёртвой зоны
         Min : Real;   // Нижняя граница мёртвой зоны
      END_STRUCT;
   END_VAR
   VAR
      Converter : "Converter_LAD";   // Конвертер выхода
      Conveter_Back : "Converter_LAD";   // Конвертер Hand_SP в 0..100
   END_VAR
   VAR DB_SPECIFIC
      pos { S7_SetPoint := 'True'} : Array[0..15] of Bool;
   END_VAR
   VAR_TEMP
      x0 : Real;
   END_VAR
   // CMD.Start_A := true;
   VAR_TEMP   // added for the SCL form of the ladder/FBD networks
      _w1 : Bool;
      _w2 : Bool;
      _w3 : Bool;
      _w4 : Bool;
      _w5 : Bool;
      _w6 : Bool;
      _w7 : Bool;
   END_VAR
BEGIN

REGION Network 1: Сброс ПИД
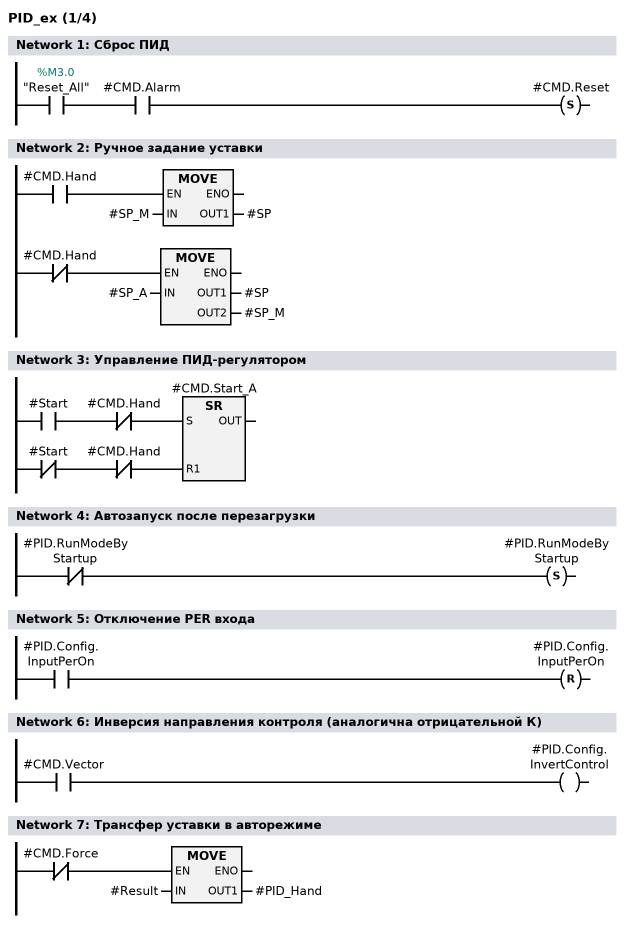
   RUNG wire#powerrail
      Contact( "Reset_All" )
      Contact( #CMD.Alarm )
      S_Coil( #CMD.Reset )
   END_RUNG
   // the same network as SCL:
   IF "Reset_All" AND #CMD.Alarm THEN #CMD.Reset := TRUE; END_IF;
END_REGION

REGION Network 2: Ручное задание уставки
   RUNG wire#powerrail
      Contact( #CMD.Hand )
      Move(in := #SP_M, out1 => #SP)
   END_RUNG
   RUNG wire#powerrail
      I_Contact( #CMD.Hand )
      Move(in := #SP_A, out1 => #SP, out2 => #SP_M)
   END_RUNG
   // the same network as SCL:
   IF #CMD.Hand THEN #SP := #SP_M; END_IF;
   IF NOT #CMD.Hand THEN
       #SP := #SP_A;
       #SP_M := #SP_A;
   END_IF;
END_REGION

REGION Network 3: Управление ПИД-регулятором
   RUNG wire#powerrail
      Contact( #Start )
      I_Contact( #CMD.Hand )
      S_SR(operand := #CMD.Start_A, r1 := wire#w1)
   END_RUNG
   RUNG wire#powerrail
      I_Contact( #Start )
      I_Contact( #CMD.Hand )
   END_RUNG wire#w1
   // the same network as SCL:
   IF #Start AND NOT #CMD.Hand THEN
       #CMD.Start_A := TRUE;   // SR flip-flop
   END_IF;
   IF NOT #Start AND NOT #CMD.Hand THEN #CMD.Start_A := FALSE; END_IF;
END_REGION

REGION Network 4: Автозапуск после перезагрузки
   RUNG wire#powerrail
      I_Contact( #PID.RunModeByStartup )
      S_Coil( #PID.RunModeByStartup )
   END_RUNG
   // the same network as SCL:
   IF NOT #PID.RunModeByStartup THEN #PID.RunModeByStartup := TRUE; END_IF;
END_REGION

REGION Network 5: Отключение PER входа
   RUNG wire#powerrail
      Contact( #PID.Config.InputPerOn )
      R_Coil( #PID.Config.InputPerOn )
   END_RUNG
   // the same network as SCL:
   IF #PID.Config.InputPerOn THEN #PID.Config.InputPerOn := FALSE; END_IF;
END_REGION

REGION Network 6: Инверсия направления контроля (аналогична отрицательной К)
   RUNG wire#powerrail
      Contact( #CMD.Vector )
      Coil( #PID.Config.InvertControl )
   END_RUNG
   // the same network as SCL:
   #PID.Config.InvertControl := #CMD.Vector;
END_REGION

REGION Network 7: Трансфер уставки в авторежиме
   RUNG wire#powerrail
      I_Contact( #CMD.Force )
      Move(in := #Result, out1 => #PID_Hand)
   END_RUNG
   // the same network as SCL:
   IF NOT #CMD.Force THEN #PID_Hand := #Result; END_IF;
END_REGION

REGION Network 8: Активация после смены режима
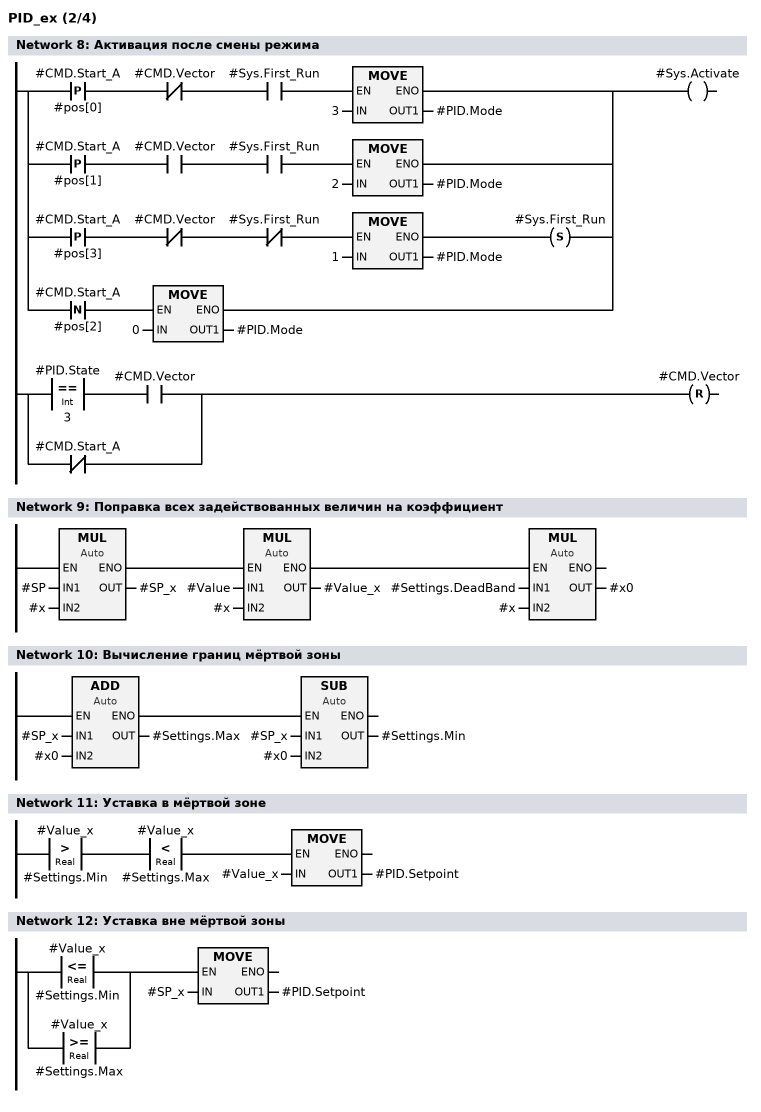
   RUNG wire#powerrail
      P_Contact(operand := #CMD.Start_A, bit := #pos[0])
      I_Contact( #CMD.Vector )
      Contact( #Sys.First_Run )
      Move(in := 3, out1 => #PID.Mode)
      wire#w1
      Coil( #Sys.Activate )
   END_RUNG
   RUNG wire#powerrail
      P_Contact(operand := #CMD.Start_A, bit := #pos[1])
      Contact( #CMD.Vector )
      Contact( #Sys.First_Run )
      Move(in := 2, out1 => #PID.Mode)
   END_RUNG wire#w1
   RUNG wire#powerrail
      P_Contact(operand := #CMD.Start_A, bit := #pos[3])
      I_Contact( #CMD.Vector )
      I_Contact( #Sys.First_Run )
      Move(in := 1, out1 => #PID.Mode)
      S_Coil( #Sys.First_Run )
   END_RUNG wire#w1
   RUNG wire#powerrail
      N_Contact(operand := #CMD.Start_A, bit := #pos[2])
      Move(in := 0, out1 => #PID.Mode)
   END_RUNG wire#w1
   RUNG wire#powerrail
      { S7_Templates := "SrcType := Int" } EQ_Contact(in1 := #PID.State, in2 := 3)
      Contact( #CMD.Vector )
      wire#w2
      R_Coil( #CMD.Vector )
   END_RUNG
   RUNG wire#powerrail
      I_Contact( #CMD.Start_A )
   END_RUNG wire#w2
   // the same network as SCL:
   #_w1 := #CMD.Start_A AND NOT #pos[0];   // rising edge of #CMD.Start_A
   #pos[0] := #CMD.Start_A;
   #_w2 := #_w1 AND NOT #CMD.Vector AND #Sys.First_Run;
   IF #_w2 THEN #PID.Mode := 3; END_IF;
   #_w3 := #CMD.Start_A AND NOT #pos[1];   // rising edge of #CMD.Start_A
   #pos[1] := #CMD.Start_A;
   #_w4 := #_w3 AND #CMD.Vector AND #Sys.First_Run;
   IF #_w4 THEN #PID.Mode := 2; END_IF;
   #_w5 := #CMD.Start_A AND NOT #pos[3];   // rising edge of #CMD.Start_A
   #pos[3] := #CMD.Start_A;
   #_w6 := #_w5 AND NOT #CMD.Vector AND NOT #Sys.First_Run;
   IF #_w6 THEN
       #PID.Mode := 1;
       #Sys.First_Run := TRUE;
   END_IF;
   #_w7 := NOT #CMD.Start_A AND #pos[2];   // falling edge of #CMD.Start_A
   #pos[2] := #CMD.Start_A;
   IF #_w7 THEN #PID.Mode := 0; END_IF;
   #Sys.Activate := #_w2 OR #_w4 OR #_w6 OR #_w7;
   IF ((#PID.State = 3) AND #CMD.Vector) OR NOT #CMD.Start_A THEN #CMD.Vector := FALSE; END_IF;
END_REGION

REGION Network 9: Поправка всех задействованных величин на коэффициент
   RUNG wire#powerrail
      Mul(in1 := #SP, in2 := #x, out => #SP_x)
      Mul(in1 := #Value, in2 := #x, out => #Value_x)
      Mul(in1 := #Settings.DeadBand, in2 := #x, out => #x0)
   END_RUNG
   // the same network as SCL:
   #SP_x := #SP * #x;
   #Value_x := #Value * #x;
   #x0 := #Settings.DeadBand * #x;
END_REGION

REGION Network 10: Вычисление границ мёртвой зоны
   RUNG wire#powerrail
      Add(in1 := #SP_x, in2 := #x0, out => #Settings.Max)
      Sub(in1 := #SP_x, in2 := #x0, out => #Settings.Min)
   END_RUNG
   // the same network as SCL:
   #Settings.Max := #SP_x + #x0;
   #Settings.Min := #SP_x - #x0;
END_REGION

REGION Network 11: Уставка в мёртвой зоне
   RUNG wire#powerrail
      { S7_Templates := "SrcType := Real" } GT_Contact(in1 := #Value_x, in2 := #Settings.Min)
      { S7_Templates := "SrcType := Real" } LT_Contact(in1 := #Value_x, in2 := #Settings.Max)
      Move(in := #Value_x, out1 => #PID.Setpoint)
   END_RUNG
   // the same network as SCL:
   IF (#Value_x > #Settings.Min) AND (#Value_x < #Settings.Max) THEN #PID.Setpoint := #Value_x; END_IF;
END_REGION

REGION Network 12: Уставка вне мёртвой зоны
   RUNG wire#powerrail
      { S7_Templates := "SrcType := Real" } LE_Contact(in1 := #Value_x, in2 := #Settings.Min)
      wire#w1
      Move(in := #SP_x, out1 => #PID.Setpoint)
   END_RUNG
   RUNG wire#powerrail
      { S7_Templates := "SrcType := Real" } GE_Contact(in1 := #Value_x, in2 := #Settings.Max)
   END_RUNG wire#w1
   // the same network as SCL:
   IF (#Value_x <= #Settings.Min) OR (#Value_x >= #Settings.Max) THEN #PID.Setpoint := #SP_x; END_IF;
END_REGION

REGION Network 13: ПИД
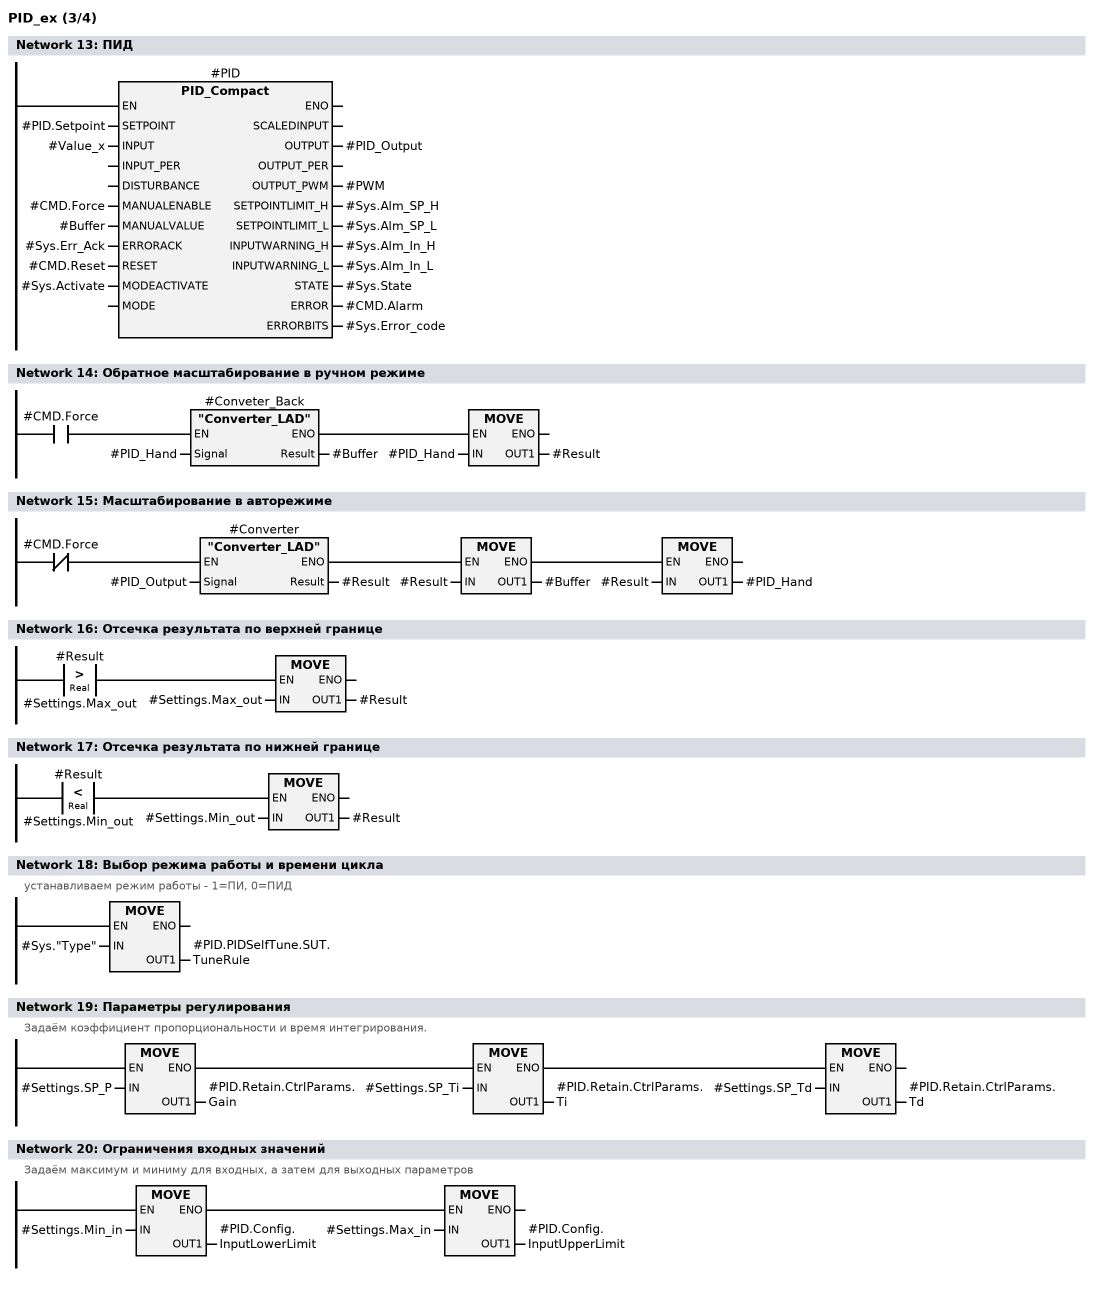
   RUNG wire#powerrail
      #PID.PID_Compact(Setpoint := #PID.Setpoint, Input := #Value_x, Input_PER :=, Disturbance :=, ManualEnable := #CMD.Force, ManualValue := #Buffer, ErrorAck := #Sys.Err_Ack, Reset := #CMD.Reset, ModeActivate := #Sys.Activate, Mode :=, ScaledInput =>, Output => #PID_Output, Output_PER =>, Output_PWM => #PWM, SetpointLimit_H => #Sys.Alm_SP_H, SetpointLimit_L => #Sys.Alm_SP_L, InputWarning_H => #Sys.Alm_In_H, InputWarning_L => #Sys.Alm_In_L, State => #Sys.State, Error => #CMD.Alarm, ErrorBits => #Sys.Error_code)
   END_RUNG
   // the same network as SCL:
   #PID(Setpoint := #PID.Setpoint,   // PID_Compact
        Input := #Value_x,
        ManualEnable := #CMD.Force,
        ManualValue := #Buffer,
        ErrorAck := #Sys.Err_Ack,
        Reset := #CMD.Reset,
        ModeActivate := #Sys.Activate,
        Output => #PID_Output,
        Output_PWM => #PWM,
        SetpointLimit_H => #Sys.Alm_SP_H,
        SetpointLimit_L => #Sys.Alm_SP_L,
        InputWarning_H => #Sys.Alm_In_H,
        InputWarning_L => #Sys.Alm_In_L,
        State => #Sys.State,
        Error => #CMD.Alarm,
        ErrorBits => #Sys.Error_code);
END_REGION

REGION Network 14: Обратное масштабирование в ручном режиме
   RUNG wire#powerrail
      Contact( #CMD.Force )
      #Conveter_Back(Signal := #PID_Hand, Result => #Buffer)
      { S7_GenerateENO := "TRUE" } Move(in := #PID_Hand, out1 => #Result)
   END_RUNG
   // the same network as SCL:
   #Conveter_Back(EN := #CMD.Force, Signal := #PID_Hand, Result => #Buffer, ENO => #_w1);   // "Converter_LAD"
   IF #_w1 THEN #Result := #PID_Hand; END_IF;
END_REGION

REGION Network 15: Масштабирование в авторежиме
   RUNG wire#powerrail
      I_Contact( #CMD.Force )
      #Converter(Signal := #PID_Output, Result => #Result)
      { S7_GenerateENO := "TRUE" } Move(in := #Result, out1 => #Buffer)
      { S7_GenerateENO := "TRUE" } Move(in := #Result, out1 => #PID_Hand)
   END_RUNG
   // the same network as SCL:
   // ENO of a box is taken as its EN; it also drops when the box reports an error
   #Converter(EN := NOT #CMD.Force, Signal := #PID_Output, Result => #Result, ENO => #_w1);   // "Converter_LAD"
   IF #_w1 THEN
       #Buffer := #Result;
       #PID_Hand := #Result;
   END_IF;
END_REGION

REGION Network 16: Отсечка результата по верхней границе
   RUNG wire#powerrail
      { S7_Templates := "SrcType := Real" } GT_Contact(in1 := #Result, in2 := #Settings.Max_out)
      Move(in := #Settings.Max_out, out1 => #Result)
   END_RUNG
   // the same network as SCL:
   IF #Result > #Settings.Max_out THEN #Result := #Settings.Max_out; END_IF;
END_REGION

REGION Network 17: Отсечка результата по нижней границе
   RUNG wire#powerrail
      { S7_Templates := "SrcType := Real" } LT_Contact(in1 := #Result, in2 := #Settings.Min_out)
      Move(in := #Settings.Min_out, out1 => #Result)
   END_RUNG
   // the same network as SCL:
   IF #Result < #Settings.Min_out THEN #Result := #Settings.Min_out; END_IF;
END_REGION

REGION Network 18: Выбор режима работы и времени цикла
   // устанавливаем режим работы - 1=ПИ, 0=ПИД
   RUNG wire#powerrail
      { S7_GenerateENO := "TRUE" } Move(in := #Sys."Type", out1 => #PID.PIDSelfTune.SUT.TuneRule)
   END_RUNG
   // the same network as SCL:
   #PID.PIDSelfTune.SUT.TuneRule := #Sys."Type";
END_REGION

REGION Network 19: Параметры регулирования
   // Задаём коэффициент пропорциональности и время интегрирования.
   RUNG wire#powerrail
      { S7_GenerateENO := "TRUE" } Move(in := #Settings.SP_P, out1 => #PID.Retain.CtrlParams.Gain)
      { S7_GenerateENO := "TRUE" } Move(in := #Settings.SP_Ti, out1 => #PID.Retain.CtrlParams.Ti)
      { S7_GenerateENO := "TRUE" } Move(in := #Settings.SP_Td, out1 => #PID.Retain.CtrlParams.Td)
   END_RUNG
   // the same network as SCL:
   // ENO of a box is taken as its EN; it also drops when the box reports an error
   #PID.Retain.CtrlParams.Gain := #Settings.SP_P;
   #PID.Retain.CtrlParams.Ti := #Settings.SP_Ti;
   #PID.Retain.CtrlParams.Td := #Settings.SP_Td;
END_REGION

REGION Network 20: Ограничения входных значений
   // Задаём максимум и миниму для входных, а затем для выходных параметров
   RUNG wire#powerrail
      { S7_GenerateENO := "TRUE" } Move(in := #Settings.Min_in, out1 => #PID.Config.InputLowerLimit)
      { S7_GenerateENO := "TRUE" } Move(in := #Settings.Max_in, out1 => #PID.Config.InputUpperLimit)
   END_RUNG
   // the same network as SCL:
   // ENO of a box is taken as its EN; it also drops when the box reports an error
   #PID.Config.InputLowerLimit := #Settings.Min_in;
   #PID.Config.InputUpperLimit := #Settings.Max_in;
END_REGION

REGION Network 21: Ограничения выходных значений
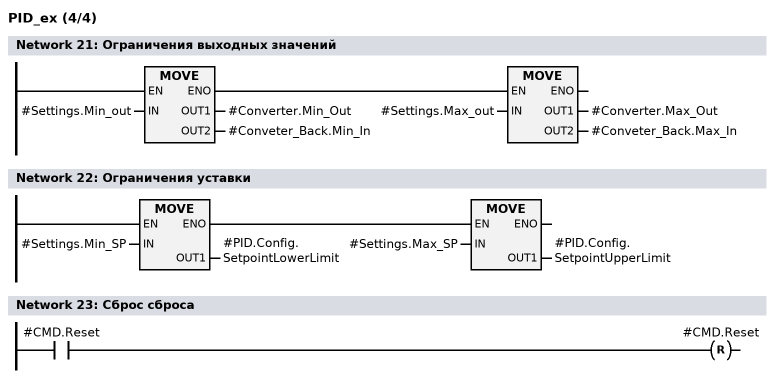
   RUNG wire#powerrail
      { S7_GenerateENO := "TRUE" } Move(in := #Settings.Min_out, out1 => #Converter.Min_Out, out2 => #Conveter_Back.Min_In)
      { S7_GenerateENO := "TRUE" } Move(in := #Settings.Max_out, out1 => #Converter.Max_Out, out2 => #Conveter_Back.Max_In)
   END_RUNG
   // the same network as SCL:
   // ENO of a box is taken as its EN; it also drops when the box reports an error
   #Converter.Min_Out := #Settings.Min_out;
   #Conveter_Back.Min_In := #Settings.Min_out;
   #Converter.Max_Out := #Settings.Max_out;
   #Conveter_Back.Max_In := #Settings.Max_out;
END_REGION

REGION Network 22: Ограничения уставки
   RUNG wire#powerrail
      { S7_GenerateENO := "TRUE" } Move(in := #Settings.Min_SP, out1 => #PID.Config.SetpointLowerLimit)
      { S7_GenerateENO := "TRUE" } Move(in := #Settings.Max_SP, out1 => #PID.Config.SetpointUpperLimit)
   END_RUNG
   // the same network as SCL:
   // ENO of a box is taken as its EN; it also drops when the box reports an error
   #PID.Config.SetpointLowerLimit := #Settings.Min_SP;
   #PID.Config.SetpointUpperLimit := #Settings.Max_SP;
END_REGION

REGION Network 23: Сброс сброса
   RUNG wire#powerrail
      Contact( #CMD.Reset )
      R_Coil( #CMD.Reset )
   END_RUNG
   // the same network as SCL:
   IF #CMD.Reset THEN #CMD.Reset := FALSE; END_IF;
END_REGION
END_FUNCTION_BLOCK

ORGANIZATION_BLOCK "Diagnostic error interrupt"   // OB82, LAD, DiagnosticErrorInterrupt
{ S7_Optimized_Access := 'TRUE' }
VERSION : 0.1
// stored: IsIECCheckEnabled false, SetENOAutomatically false
   VAR_INPUT
      IO_State : Word;   // IO state of the HW object
      LADDR : HW_ANY;   // Hardware identifier
      Channel : UInt;   // Channel number
      MultiError : Bool;   // =true if more than one error is present
   END_VAR
BEGIN
END_ORGANIZATION_BLOCK

ORGANIZATION_BLOCK "Programming error"   // OB121, LAD, ProgrammingError
{ S7_Optimized_Access := 'TRUE' }
VERSION : 0.1
// stored: IsIECCheckEnabled false, SetENOAutomatically false
   VAR_INPUT
      BlockNr : UInt;   // Number of causing block
      Reaction : USInt;   // 0:ignore, 1:substitute, 2:skip
      Fault_ID : Byte;   // Fault identifier
      BlockType : USInt;   // 16#01:OB, 16#02:FC, 16#03:FB, 16#04:SFC, 16#05:SFB, 16#06:DB: Type of block causing the error
      Area : USInt;   // Area where the error occured
      DBNr : DB_ANY;   // DB number if Area = DB or DI
      Csg_OBNr : OB_ANY;   // Number of OB causing the error
      Csg_Prio : USInt;   // Priority of OB causing the error
      Width : USInt;   // 0:bit, 1:byte, 2:word, 3:dword, 4:lword
   END_VAR
BEGIN
END_ORGANIZATION_BLOCK

ORGANIZATION_BLOCK "Pull or plug of modules"   // OB83, LAD, PullOrPlugOfModules
{ S7_Optimized_Access := 'TRUE' }
VERSION : 0.1
// stored: IsIECCheckEnabled false, SetENOAutomatically false
   VAR_INPUT
      LADDR : HW_IO;   // Hardware identifier
      Event_Class : Byte;   // 16#38/39: module inserted, removed
      Fault_ID : Byte;   // Fault identifier
   END_VAR
BEGIN
END_ORGANIZATION_BLOCK

ORGANIZATION_BLOCK "Rack or station failure"   // OB86, LAD, RackOrStationFailure
{ S7_Optimized_Access := 'TRUE' }
VERSION : 0.1
// stored: IsIECCheckEnabled false, SetENOAutomatically false
   VAR_INPUT
      LADDR : HW_DEVICE;   // Hardware identifier
      Event_Class : Byte;   // Event class
      Fault_ID : Byte;   // Fault identifier
   END_VAR
BEGIN
END_ORGANIZATION_BLOCK

FUNCTION_BLOCK "Route_Check"   // FB3, LAD
TITLE = Проверка маршрутов для заполнения РВ
{ S7_Optimized_Access := 'TRUE' }
VERSION : 0.1
// stored: AutoNumber true, IsIECCheckEnabled false, IsRetainMemResEnabled false, MemoryReserve 100, SetENOAutomatically false, UDAEnableTagReadback false
   VAR
      ready_2_7_from_2_9 : Bool;
      ready_2_7_from_SKV13 : Bool;
      ready_2_7_from_2_6_1 : Bool;
      ready_2_7_from_2_6_2 : Bool;
      ready_2_7_q_1 : Bool;
      ready_2_7_q_2 : Bool;
      ready_2_6_from_SKV14 : Bool;
      ready_2_6_from_2_5_1 : Bool;
      ready_2_6_from_2_5_2 : Bool;
      ready_2_6_q_1 : Bool;
      ready_2_6_q_2 : Bool;
   END_VAR
BEGIN

REGION Network 1: СКВ-2
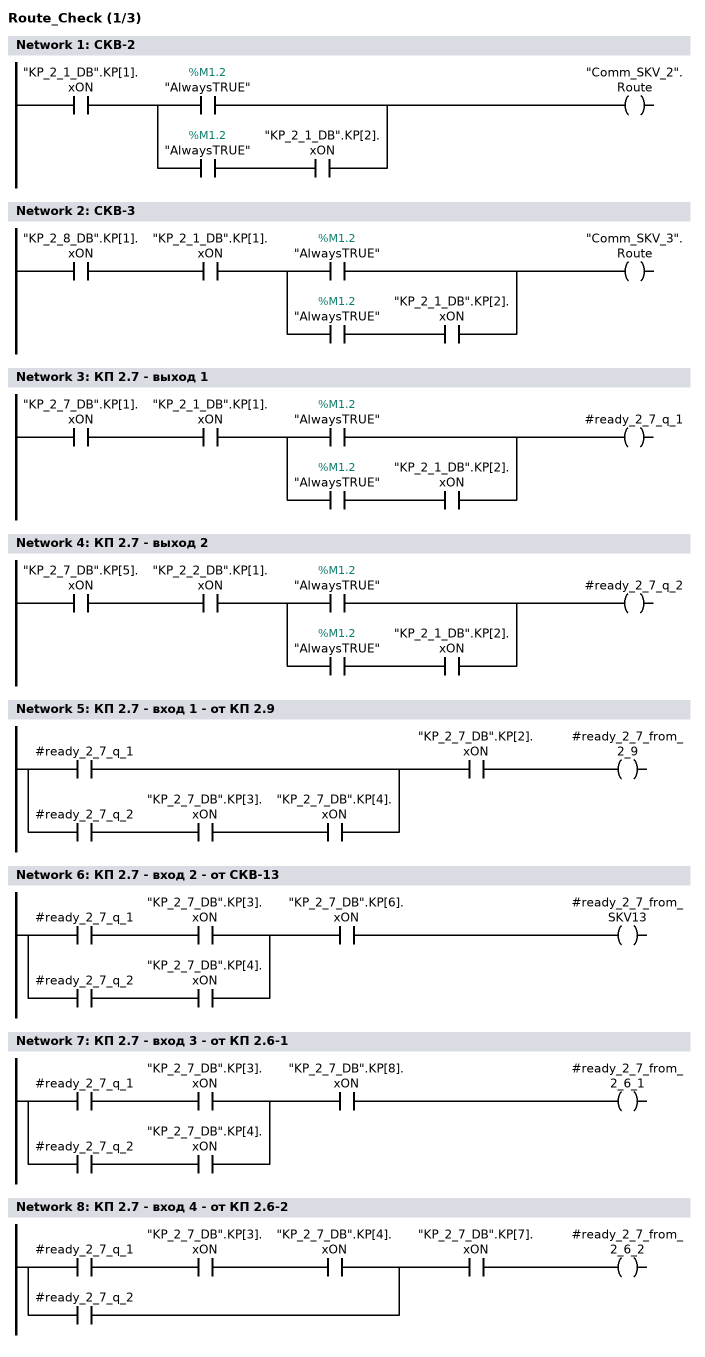
   RUNG wire#powerrail
      Contact( "KP_2_1_DB".KP[1].xON )
      wire#w1
      Contact( "AlwaysTRUE" )
      wire#w2
      Coil( "Comm_SKV_2".Route )
   END_RUNG
   RUNG wire#w1
      Contact( "AlwaysTRUE" )
      Contact( "KP_2_1_DB".KP[2].xON )
   END_RUNG wire#w2
   // the same network as SCL:
   "Comm_SKV_2".Route := "KP_2_1_DB".KP[1].xON AND ("AlwaysTRUE" OR ("AlwaysTRUE" AND "KP_2_1_DB".KP[2].xON));
END_REGION

REGION Network 2: СКВ-3
   RUNG wire#powerrail
      Contact( "KP_2_8_DB".KP[1].xON )
      Contact( "KP_2_1_DB".KP[1].xON )
      wire#w1
      Contact( "AlwaysTRUE" )
      wire#w2
      Coil( "Comm_SKV_3".Route )
   END_RUNG
   RUNG wire#w1
      Contact( "AlwaysTRUE" )
      Contact( "KP_2_1_DB".KP[2].xON )
   END_RUNG wire#w2
   // the same network as SCL:
   "Comm_SKV_3".Route := "KP_2_8_DB".KP[1].xON AND "KP_2_1_DB".KP[1].xON AND ("AlwaysTRUE" OR ("AlwaysTRUE" AND "KP_2_1_DB".KP[2].xON));
END_REGION

REGION Network 3: КП 2.7 - выход 1
   RUNG wire#powerrail
      Contact( "KP_2_7_DB".KP[1].xON )
      Contact( "KP_2_1_DB".KP[1].xON )
      wire#w1
      Contact( "AlwaysTRUE" )
      wire#w2
      Coil( #ready_2_7_q_1 )
   END_RUNG
   RUNG wire#w1
      Contact( "AlwaysTRUE" )
      Contact( "KP_2_1_DB".KP[2].xON )
   END_RUNG wire#w2
   // the same network as SCL:
   #ready_2_7_q_1 := "KP_2_7_DB".KP[1].xON AND "KP_2_1_DB".KP[1].xON AND ("AlwaysTRUE" OR ("AlwaysTRUE" AND "KP_2_1_DB".KP[2].xON));
END_REGION

REGION Network 4: КП 2.7 - выход 2
   RUNG wire#powerrail
      Contact( "KP_2_7_DB".KP[5].xON )
      Contact( "KP_2_2_DB".KP[1].xON )
      wire#w1
      Contact( "AlwaysTRUE" )
      wire#w2
      Coil( #ready_2_7_q_2 )
   END_RUNG
   RUNG wire#w1
      Contact( "AlwaysTRUE" )
      Contact( "KP_2_1_DB".KP[2].xON )
   END_RUNG wire#w2
   // the same network as SCL:
   #ready_2_7_q_2 := "KP_2_7_DB".KP[5].xON AND "KP_2_2_DB".KP[1].xON AND ("AlwaysTRUE" OR ("AlwaysTRUE" AND "KP_2_1_DB".KP[2].xON));
END_REGION

REGION Network 5: КП 2.7 - вход 1 - от КП 2.9
   RUNG wire#powerrail
      Contact( #ready_2_7_q_1 )
      wire#w1
      Contact( "KP_2_7_DB".KP[2].xON )
      Coil( #ready_2_7_from_2_9 )
   END_RUNG
   RUNG wire#powerrail
      Contact( #ready_2_7_q_2 )
      Contact( "KP_2_7_DB".KP[3].xON )
      Contact( "KP_2_7_DB".KP[4].xON )
   END_RUNG wire#w1
   // the same network as SCL:
   #ready_2_7_from_2_9 := (#ready_2_7_q_1 OR (#ready_2_7_q_2 AND "KP_2_7_DB".KP[3].xON AND "KP_2_7_DB".KP[4].xON)) AND "KP_2_7_DB".KP[2].xON;
END_REGION

REGION Network 6: КП 2.7 - вход 2 - от СКВ-13
   RUNG wire#powerrail
      Contact( #ready_2_7_q_1 )
      Contact( "KP_2_7_DB".KP[3].xON )
      wire#w1
      Contact( "KP_2_7_DB".KP[6].xON )
      Coil( #ready_2_7_from_SKV13 )
   END_RUNG
   RUNG wire#powerrail
      Contact( #ready_2_7_q_2 )
      Contact( "KP_2_7_DB".KP[4].xON )
   END_RUNG wire#w1
   // the same network as SCL:
   #ready_2_7_from_SKV13 := ((#ready_2_7_q_1 AND "KP_2_7_DB".KP[3].xON) OR (#ready_2_7_q_2 AND "KP_2_7_DB".KP[4].xON)) AND "KP_2_7_DB".KP[6].xON;
END_REGION

REGION Network 7: КП 2.7 - вход 3 - от КП 2.6-1
   RUNG wire#powerrail
      Contact( #ready_2_7_q_1 )
      Contact( "KP_2_7_DB".KP[3].xON )
      wire#w1
      Contact( "KP_2_7_DB".KP[8].xON )
      Coil( #ready_2_7_from_2_6_1 )
   END_RUNG
   RUNG wire#powerrail
      Contact( #ready_2_7_q_2 )
      Contact( "KP_2_7_DB".KP[4].xON )
   END_RUNG wire#w1
   // the same network as SCL:
   #ready_2_7_from_2_6_1 := ((#ready_2_7_q_1 AND "KP_2_7_DB".KP[3].xON) OR (#ready_2_7_q_2 AND "KP_2_7_DB".KP[4].xON)) AND "KP_2_7_DB".KP[8].xON;
END_REGION

REGION Network 8: КП 2.7 - вход 4 - от КП 2.6-2
   RUNG wire#powerrail
      Contact( #ready_2_7_q_1 )
      Contact( "KP_2_7_DB".KP[3].xON )
      Contact( "KP_2_7_DB".KP[4].xON )
      wire#w1
      Contact( "KP_2_7_DB".KP[7].xON )
      Coil( #ready_2_7_from_2_6_2 )
   END_RUNG
   RUNG wire#powerrail
      Contact( #ready_2_7_q_2 )
   END_RUNG wire#w1
   // the same network as SCL:
   #ready_2_7_from_2_6_2 := ((#ready_2_7_q_1 AND "KP_2_7_DB".KP[3].xON AND "KP_2_7_DB".KP[4].xON) OR #ready_2_7_q_2) AND "KP_2_7_DB".KP[7].xON;
END_REGION

REGION Network 9: СКВ-23
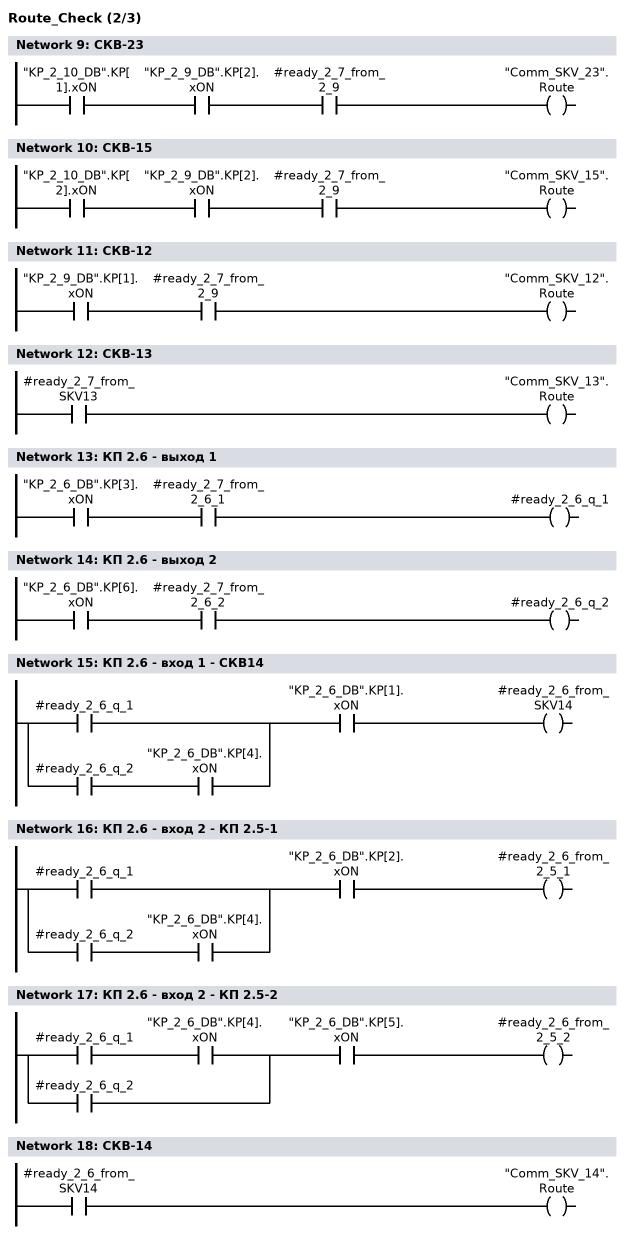
   RUNG wire#powerrail
      Contact( "KP_2_10_DB".KP[1].xON )
      Contact( "KP_2_9_DB".KP[2].xON )
      Contact( #ready_2_7_from_2_9 )
      Coil( "Comm_SKV_23".Route )
   END_RUNG
   // the same network as SCL:
   "Comm_SKV_23".Route := "KP_2_10_DB".KP[1].xON AND "KP_2_9_DB".KP[2].xON AND #ready_2_7_from_2_9;
END_REGION

REGION Network 10: СКВ-15
   RUNG wire#powerrail
      Contact( "KP_2_10_DB".KP[2].xON )
      Contact( "KP_2_9_DB".KP[2].xON )
      Contact( #ready_2_7_from_2_9 )
      Coil( "Comm_SKV_15".Route )
   END_RUNG
   // the same network as SCL:
   "Comm_SKV_15".Route := "KP_2_10_DB".KP[2].xON AND "KP_2_9_DB".KP[2].xON AND #ready_2_7_from_2_9;
END_REGION

REGION Network 11: СКВ-12
   RUNG wire#powerrail
      Contact( "KP_2_9_DB".KP[1].xON )
      Contact( #ready_2_7_from_2_9 )
      Coil( "Comm_SKV_12".Route )
   END_RUNG
   // the same network as SCL:
   "Comm_SKV_12".Route := "KP_2_9_DB".KP[1].xON AND #ready_2_7_from_2_9;
END_REGION

REGION Network 12: СКВ-13
   RUNG wire#powerrail
      Contact( #ready_2_7_from_SKV13 )
      Coil( "Comm_SKV_13".Route )
   END_RUNG
   // the same network as SCL:
   "Comm_SKV_13".Route := #ready_2_7_from_SKV13;
END_REGION

REGION Network 13: КП 2.6 - выход 1
   RUNG wire#powerrail
      Contact( "KP_2_6_DB".KP[3].xON )
      Contact( #ready_2_7_from_2_6_1 )
      Coil( #ready_2_6_q_1 )
   END_RUNG
   // the same network as SCL:
   #ready_2_6_q_1 := "KP_2_6_DB".KP[3].xON AND #ready_2_7_from_2_6_1;
END_REGION

REGION Network 14: КП 2.6 - выход 2
   RUNG wire#powerrail
      Contact( "KP_2_6_DB".KP[6].xON )
      Contact( #ready_2_7_from_2_6_2 )
      Coil( #ready_2_6_q_2 )
   END_RUNG
   // the same network as SCL:
   #ready_2_6_q_2 := "KP_2_6_DB".KP[6].xON AND #ready_2_7_from_2_6_2;
END_REGION

REGION Network 15: КП 2.6 - вход 1 - СКВ14
   RUNG wire#powerrail
      Contact( #ready_2_6_q_1 )
      wire#w1
      Contact( "KP_2_6_DB".KP[1].xON )
      Coil( #ready_2_6_from_SKV14 )
   END_RUNG
   RUNG wire#powerrail
      Contact( #ready_2_6_q_2 )
      Contact( "KP_2_6_DB".KP[4].xON )
   END_RUNG wire#w1
   // the same network as SCL:
   #ready_2_6_from_SKV14 := (#ready_2_6_q_1 OR (#ready_2_6_q_2 AND "KP_2_6_DB".KP[4].xON)) AND "KP_2_6_DB".KP[1].xON;
END_REGION

REGION Network 16: КП 2.6 - вход 2 - КП 2.5-1
   RUNG wire#powerrail
      Contact( #ready_2_6_q_1 )
      wire#w1
      Contact( "KP_2_6_DB".KP[2].xON )
      Coil( #ready_2_6_from_2_5_1 )
   END_RUNG
   RUNG wire#powerrail
      Contact( #ready_2_6_q_2 )
      Contact( "KP_2_6_DB".KP[4].xON )
   END_RUNG wire#w1
   // the same network as SCL:
   #ready_2_6_from_2_5_1 := (#ready_2_6_q_1 OR (#ready_2_6_q_2 AND "KP_2_6_DB".KP[4].xON)) AND "KP_2_6_DB".KP[2].xON;
END_REGION

REGION Network 17: КП 2.6 - вход 2 - КП 2.5-2
   RUNG wire#powerrail
      Contact( #ready_2_6_q_1 )
      Contact( "KP_2_6_DB".KP[4].xON )
      wire#w1
      Contact( "KP_2_6_DB".KP[5].xON )
      Coil( #ready_2_6_from_2_5_2 )
   END_RUNG
   RUNG wire#powerrail
      Contact( #ready_2_6_q_2 )
   END_RUNG wire#w1
   // the same network as SCL:
   #ready_2_6_from_2_5_2 := ((#ready_2_6_q_1 AND "KP_2_6_DB".KP[4].xON) OR #ready_2_6_q_2) AND "KP_2_6_DB".KP[5].xON;
END_REGION

REGION Network 18: СКВ-14
   RUNG wire#powerrail
      Contact( #ready_2_6_from_SKV14 )
      Coil( "Comm_SKV_14".Route )
   END_RUNG
   // the same network as SCL:
   "Comm_SKV_14".Route := #ready_2_6_from_SKV14;
END_REGION

REGION Network 19: СКВ-1
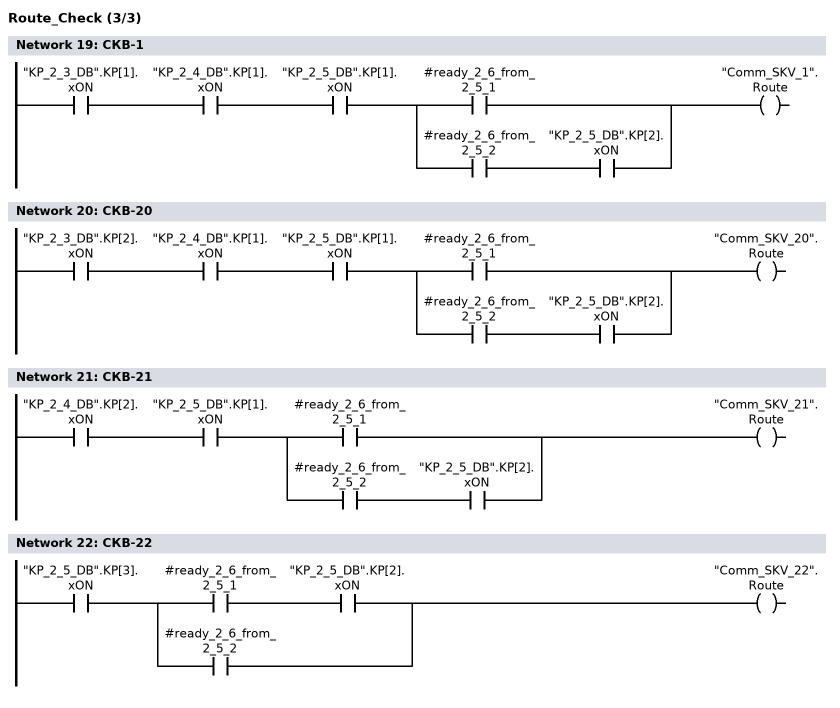
   RUNG wire#powerrail
      Contact( "KP_2_3_DB".KP[1].xON )
      Contact( "KP_2_4_DB".KP[1].xON )
      Contact( "KP_2_5_DB".KP[1].xON )
      wire#w1
      Contact( #ready_2_6_from_2_5_1 )
      wire#w2
      Coil( "Comm_SKV_1".Route )
   END_RUNG
   RUNG wire#w1
      Contact( #ready_2_6_from_2_5_2 )
      Contact( "KP_2_5_DB".KP[2].xON )
   END_RUNG wire#w2
   // the same network as SCL:
   "Comm_SKV_1".Route := "KP_2_3_DB".KP[1].xON AND "KP_2_4_DB".KP[1].xON AND "KP_2_5_DB".KP[1].xON AND (#ready_2_6_from_2_5_1 OR (#ready_2_6_from_2_5_2 AND "KP_2_5_DB".KP[2].xON));
END_REGION

REGION Network 20: СКВ-20
   RUNG wire#powerrail
      Contact( "KP_2_3_DB".KP[2].xON )
      Contact( "KP_2_4_DB".KP[1].xON )
      Contact( "KP_2_5_DB".KP[1].xON )
      wire#w1
      Contact( #ready_2_6_from_2_5_1 )
      wire#w2
      Coil( "Comm_SKV_20".Route )
   END_RUNG
   RUNG wire#w1
      Contact( #ready_2_6_from_2_5_2 )
      Contact( "KP_2_5_DB".KP[2].xON )
   END_RUNG wire#w2
   // the same network as SCL:
   "Comm_SKV_20".Route := "KP_2_3_DB".KP[2].xON AND "KP_2_4_DB".KP[1].xON AND "KP_2_5_DB".KP[1].xON AND (#ready_2_6_from_2_5_1 OR (#ready_2_6_from_2_5_2 AND "KP_2_5_DB".KP[2].xON));
END_REGION

REGION Network 21: СКВ-21
   RUNG wire#powerrail
      Contact( "KP_2_4_DB".KP[2].xON )
      Contact( "KP_2_5_DB".KP[1].xON )
      wire#w1
      Contact( #ready_2_6_from_2_5_1 )
      wire#w2
      Coil( "Comm_SKV_21".Route )
   END_RUNG
   RUNG wire#w1
      Contact( #ready_2_6_from_2_5_2 )
      Contact( "KP_2_5_DB".KP[2].xON )
   END_RUNG wire#w2
   // the same network as SCL:
   "Comm_SKV_21".Route := "KP_2_4_DB".KP[2].xON AND "KP_2_5_DB".KP[1].xON AND (#ready_2_6_from_2_5_1 OR (#ready_2_6_from_2_5_2 AND "KP_2_5_DB".KP[2].xON));
END_REGION

REGION Network 22: СКВ-22
   RUNG wire#powerrail
      Contact( "KP_2_5_DB".KP[3].xON )
      wire#w1
      Contact( #ready_2_6_from_2_5_1 )
      Contact( "KP_2_5_DB".KP[2].xON )
      wire#w2
      Coil( "Comm_SKV_22".Route )
   END_RUNG
   RUNG wire#w1
      Contact( #ready_2_6_from_2_5_2 )
   END_RUNG wire#w2
   // the same network as SCL:
   "Comm_SKV_22".Route := "KP_2_5_DB".KP[3].xON AND ((#ready_2_6_from_2_5_1 AND "KP_2_5_DB".KP[2].xON) OR #ready_2_6_from_2_5_2);
END_REGION
END_FUNCTION_BLOCK

FUNCTION "FC_DRV_Start" : Void   // FC100, LAD
{ S7_Optimized_Access := 'FALSE' }
VERSION : 0.1
// stored: AutoNumber false, IsIECCheckEnabled false, SetENOAutomatically false, UDAEnableTagReadback false
BEGIN

REGION Network 1: Системное время
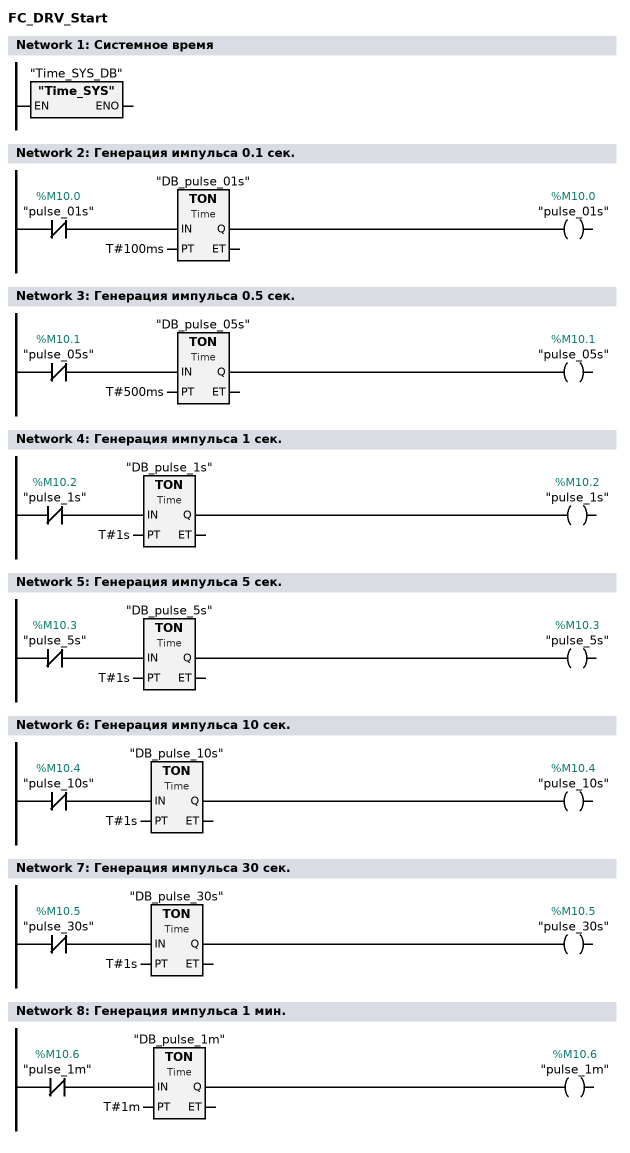
   RUNG wire#powerrail
      "Time_SYS_DB"()
   END_RUNG
   // the same network as SCL:
   "Time_SYS_DB"();   // "Time_SYS"
END_REGION

REGION Network 2: Генерация импульса 0.1 сек.
   RUNG wire#powerrail
      I_Contact( "pulse_01s" )
      { S7_Templates := "time_type := Time" } "DB_pulse_01s".TON(pt := T#100ms, et =>)
      Coil( "pulse_01s" )
   END_RUNG
   // the same network as SCL:
   "DB_pulse_01s".TON(IN := NOT "pulse_01s", PT := T#100ms);
   "pulse_01s" := "DB_pulse_01s".Q;
END_REGION

REGION Network 3: Генерация импульса 0.5 сек.
   RUNG wire#powerrail
      I_Contact( "pulse_05s" )
      { S7_Templates := "time_type := Time" } "DB_pulse_05s".TON(pt := T#500ms, et =>)
      Coil( "pulse_05s" )
   END_RUNG
   // the same network as SCL:
   "DB_pulse_05s".TON(IN := NOT "pulse_05s", PT := T#500ms);
   "pulse_05s" := "DB_pulse_05s".Q;
END_REGION

REGION Network 4: Генерация импульса 1 сек.
   RUNG wire#powerrail
      I_Contact( "pulse_1s" )
      { S7_Templates := "time_type := Time" } "DB_pulse_1s".TON(pt := T#1s, et =>)
      Coil( "pulse_1s" )
   END_RUNG
   // the same network as SCL:
   "DB_pulse_1s".TON(IN := NOT "pulse_1s", PT := T#1s);
   "pulse_1s" := "DB_pulse_1s".Q;
END_REGION

REGION Network 5: Генерация импульса 5 сек.
   RUNG wire#powerrail
      I_Contact( "pulse_5s" )
      { S7_Templates := "time_type := Time" } "DB_pulse_5s".TON(pt := T#1s, et =>)
      Coil( "pulse_5s" )
   END_RUNG
   // the same network as SCL:
   "DB_pulse_5s".TON(IN := NOT "pulse_5s", PT := T#1s);
   "pulse_5s" := "DB_pulse_5s".Q;
END_REGION

REGION Network 6: Генерация импульса 10 сек.
   RUNG wire#powerrail
      I_Contact( "pulse_10s" )
      { S7_Templates := "time_type := Time" } "DB_pulse_10s".TON(pt := T#1s, et =>)
      Coil( "pulse_10s" )
   END_RUNG
   // the same network as SCL:
   "DB_pulse_10s".TON(IN := NOT "pulse_10s", PT := T#1s);
   "pulse_10s" := "DB_pulse_10s".Q;
END_REGION

REGION Network 7: Генерация импульса 30 сек.
   RUNG wire#powerrail
      I_Contact( "pulse_30s" )
      { S7_Templates := "time_type := Time" } "DB_pulse_30s".TON(pt := T#1s, et =>)
      Coil( "pulse_30s" )
   END_RUNG
   // the same network as SCL:
   "DB_pulse_30s".TON(IN := NOT "pulse_30s", PT := T#1s);
   "pulse_30s" := "DB_pulse_30s".Q;
END_REGION

REGION Network 8: Генерация импульса 1 мин.
   RUNG wire#powerrail
      I_Contact( "pulse_1m" )
      { S7_Templates := "time_type := Time" } "DB_pulse_1m".TON(pt := T#1m, et =>)
      Coil( "pulse_1m" )
   END_RUNG
   // the same network as SCL:
   "DB_pulse_1m".TON(IN := NOT "pulse_1m", PT := T#1m);
   "pulse_1m" := "DB_pulse_1m".Q;
END_REGION
END_FUNCTION

FUNCTION_BLOCK "Historian"   // FB88, LAD
{ S7_Optimized_Access := 'FALSE' }
VERSION : 0.1
// stored: AutoNumber false, IsIECCheckEnabled false, SetENOAutomatically false, UDAEnableTagReadback false
   VAR_IN_OUT
      Main_REQ_Start : Bool;
      Main_Start : Bool;
      HMI_Start : Bool;
      HMI_Stop : Bool;
   END_VAR
   VAR DB_SPECIFIC
      pos : Array[0..15] of Bool;
      update : Bool;
      CMD : Bool;
      CODE : Int;
      DTL : DTL;
   END_VAR
   VAR
      LOG { S7_SetPoint := 'True'} : "Historian_LOG";
   END_VAR
   VAR CONSTANT
      tmp_x1 : Bool;
      tmp_x2 : Bool;
      tmp_x3 : Bool;
      any_conditions : Bool := true;
   END_VAR
   VAR_TEMP   // added for the SCL form of the ladder/FBD networks
      _w1 : Bool;
      _w2 : Bool;
      _w3 : Bool;
      _w4 : Bool;
   END_VAR
BEGIN

REGION Network 1: Запуск и останов с HMI
